//     PlcTask Inputs/GVL_iXlinker.EtherCAT_Master_ATxxxx.Beckhoff_AT1xxx.Beckhoff_AT2xxxEK1122.A_0069_AT2050_0501_0019_AT2050_0501.WcState.InputToggle <-> WcState/InputToggle
//     PlcTask Inputs/GVL_iXlinker.EtherCAT_Master_ATxxxx.Beckhoff_AT1xxx.Beckhoff_AT2xxxEK1122.A_0069_AT2050_0501_0019_AT2050_0501.InfoData.AdsAddr <-> InfoData/AdsAddr
//     PlcTask Inputs/GVL_iXlinker.EtherCAT_Master_ATxxxx.Beckhoff_AT1xxx.Beckhoff_AT2xxxEK1122.A_0069_AT2050_0501_0019_AT2050_0501.InfoData.DcOutputShift <-> InfoData/DcOutputShift
//     PlcTask Inputs/GVL_iXlinker.EtherCAT_Master_ATxxxx.Beckhoff_AT1xxx.Beckhoff_AT2xxxEK1122.A_0069_AT2050_0501_0019_AT2050_0501.InfoData.DcInputShift <-> InfoData/DcInputShift
//     PlcTask Inputs/GVL_iXlinker.EtherCAT_Master_ATxxxx.Beckhoff_AT1xxx.Beckhoff_AT2xxxEK1122.A_0069_AT2050_0501_0019_AT2050_0501.InfoData.State <-> InfoData/State
//   PLC/PLC Instance <-> EtherCAT Master ATxxxx/Beckhoff AT1xxx/Beckhoff AT2xxxEK1122/A_0069(AT2050-0501-0019) (AT2050-0501)/A_0081(AT2002-5250-0018) (AT2002-5250)
//     PlcTask Inputs/GVL_iXlinker.EtherCAT_Master_ATxxxx.Beckhoff_AT1xxx.Beckhoff_AT2xxxEK1122.A_0069_AT2050_0501_0019_AT2050_0501.A_0081_AT2002_5250_0018_AT2002_5250.FB_Inputs.Status <-> FB Inputs/Status
//     PlcTask Inputs/GVL_iXlinker.EtherCAT_Master_ATxxxx.Beckhoff_AT1xxx.Beckhoff_AT2xxxEK1122.A_0069_AT2050_0501_0019_AT2050_0501.A_0081_AT2002_5250_0018_AT2002_5250.FB_Inputs.Value_Channel[0] <-> FB Inputs/Value Channel 01
//     PlcTask Inputs/GVL_iXlinker.EtherCAT_Master_ATxxxx.Beckhoff_AT1xxx.Beckhoff_AT2xxxEK1122.A_0069_AT2050_0501_0019_AT2050_0501.A_0081_AT2002_5250_0018_AT2002_5250.FB_Inputs.Value_Channel[1] <-> FB Inputs/Value Channel 02
//     PlcTask Inputs/GVL_iXlinker.EtherCAT_Master_ATxxxx.Beckhoff_AT1xxx.Beckhoff_AT2xxxEK1122.A_0069_AT2050_0501_0019_AT2050_0501.A_0081_AT2002_5250_0018_AT2002_5250.FB_Inputs.Value_Channel[2] <-> FB Inputs/Value Channel 03
//     PlcTask Inputs/GVL_iXlinker.EtherCAT_Master_ATxxxx.Beckhoff_AT1xxx.Beckhoff_AT2xxxEK1122.A_0069_AT2050_0501_0019_AT2050_0501.A_0081_AT2002_5250_0018_AT2002_5250.FB_Inputs.Value_Channel[3] <-> FB Inputs/Value Channel 04
//     PlcTask Inputs/GVL_iXlinker.EtherCAT_Master_ATxxxx.Beckhoff_AT1xxx.Beckhoff_AT2xxxEK1122.A_0069_AT2050_0501_0019_AT2050_0501.A_0081_AT2002_5250_0018_AT2002_5250.FB_Inputs.Value_Channel[4] <-> FB Inputs/Value Channel 05
//     PlcTask Inputs/GVL_iXlinker.EtherCAT_Master_ATxxxx.Beckhoff_AT1xxx.Beckhoff_AT2xxxEK1122.A_0069_AT2050_0501_0019_AT2050_0501.A_0081_AT2002_5250_0018_AT2002_5250.FB_Inputs.Value_Channel[5] <-> FB Inputs/Value Channel 06
//     PlcTask Inputs/GVL_iXlinker.EtherCAT_Master_ATxxxx.Beckhoff_AT1xxx.Beckhoff_AT2xxxEK1122.A_0069_AT2050_0501_0019_AT2050_0501.A_0081_AT2002_5250_0018_AT2002_5250.FB_Inputs.Value_Channel[6] <-> FB Inputs/Value Channel 07
//     PlcTask Inputs/GVL_iXlinker.EtherCAT_Master_ATxxxx.Beckhoff_AT1xxx.Beckhoff_AT2xxxEK1122.A_0069_AT2050_0501_0019_AT2050_0501.A_0081_AT2002_5250_0018_AT2002_5250.FB_Inputs.Value_Channel[7] <-> FB Inputs/Value Channel 08
//     PlcTask Inputs/GVL_iXlinker.EtherCAT_Master_ATxxxx.Beckhoff_AT1xxx.Beckhoff_AT2xxxEK1122.A_0069_AT2050_0501_0019_AT2050_0501.A_0081_AT2002_5250_0018_AT2002_5250.FB_Inputs.Value_Channel[8] <-> FB Inputs/Value Channel 09
//     PlcTask Inputs/GVL_iXlinker.EtherCAT_Master_ATxxxx.Beckhoff_AT1xxx.Beckhoff_AT2xxxEK1122.A_0069_AT2050_0501_0019_AT2050_0501.A_0081_AT2002_5250_0018_AT2002_5250.FB_Inputs.Value_Channel[9] <-> FB Inputs/Value Channel 10
//     PlcTask Inputs/GVL_iXlinker.EtherCAT_Master_ATxxxx.Beckhoff_AT1xxx.Beckhoff_AT2xxxEK1122.A_0069_AT2050_0501_0019_AT2050_0501.A_0081_AT2002_5250_0018_AT2002_5250.FB_Inputs.Value_Channel[10] <-> FB Inputs/Value Channel 11
//     PlcTask Inputs/GVL_iXlinker.EtherCAT_Master_ATxxxx.Beckhoff_AT1xxx.Beckhoff_AT2xxxEK1122.A_0069_AT2050_0501_0019_AT2050_0501.A_0081_AT2002_5250_0018_AT2002_5250.FB_Inputs.Value_Channel[11] <-> FB Inputs/Value Channel 12
//     PlcTask Inputs/GVL_iXlinker.EtherCAT_Master_ATxxxx.Beckhoff_AT1xxx.Beckhoff_AT2xxxEK1122.A_0069_AT2050_0501_0019_AT2050_0501.A_0081_AT2002_5250_0018_AT2002_5250.FB_Inputs.Value_Channel[12] <-> FB Inputs/Value Channel 13
//     PlcTask Inputs/GVL_iXlinker.EtherCAT_Master_ATxxxx.Beckhoff_AT1xxx.Beckhoff_AT2xxxEK1122.A_0069_AT2050_0501_0019_AT2050_0501.A_0081_AT2002_5250_0018_AT2002_5250.FB_Inputs.Value_Channel[13] <-> FB Inputs/Value Channel 14
//     PlcTask Inputs/GVL_iXlinker.EtherCAT_Master_ATxxxx.Beckhoff_AT1xxx.Beckhoff_AT2xxxEK1122.A_0069_AT2050_0501_0019_AT2050_0501.A_0081_AT2002_5250_0018_AT2002_5250.FB_Inputs.Value_Channel[14] <-> FB Inputs/Value Channel 15
//     PlcTask Inputs/GVL_iXlinker.EtherCAT_Master_ATxxxx.Beckhoff_AT1xxx.Beckhoff_AT2xxxEK1122.A_0069_AT2050_0501_0019_AT2050_0501.A_0081_AT2002_5250_0018_AT2002_5250.FB_Inputs.Value_Channel[15] <-> FB Inputs/Value Channel 16
//     PlcTask Inputs/GVL_iXlinker.EtherCAT_Master_ATxxxx.Beckhoff_AT1xxx.Beckhoff_AT2xxxEK1122.A_0069_AT2050_0501_0019_AT2050_0501.A_0081_AT2002_5250_0018_AT2002_5250.FB_Inputs.Value_Channel[16] <-> FB Inputs/Value Channel 17
//     PlcTask Inputs/GVL_iXlinker.EtherCAT_Master_ATxxxx.Beckhoff_AT1xxx.Beckhoff_AT2xxxEK1122.A_0069_AT2050_0501_0019_AT2050_0501.A_0081_AT2002_5250_0018_AT2002_5250.FB_Inputs.Value_Channel[17] <-> FB Inputs/Value Channel 18
//     PlcTask Inputs/GVL_iXlinker.EtherCAT_Master_ATxxxx.Beckhoff_AT1xxx.Beckhoff_AT2xxxEK1122.A_0069_AT2050_0501_0019_AT2050_0501.A_0081_AT2002_5250_0018_AT2002_5250.FB_Inputs.Value_Channel[18] <-> FB Inputs/Value Channel 19
//     PlcTask Inputs/GVL_iXlinker.EtherCAT_Master_ATxxxx.Beckhoff_AT1xxx.Beckhoff_AT2xxxEK1122.A_0069_AT2050_0501_0019_AT2050_0501.A_0081_AT2002_5250_0018_AT2002_5250.FB_Inputs.Value_Channel[19] <-> FB Inputs/Value Channel 20
//     PlcTask Inputs/GVL_iXlinker.EtherCAT_Master_ATxxxx.Beckhoff_AT1xxx.Beckhoff_AT2xxxEK1122.A_0069_AT2050_0501_0019_AT2050_0501.A_0081_AT2002_5250_0018_AT2002_5250.FB_Inputs.Value_Channel[20] <-> FB Inputs/Value Channel 21
//     PlcTask Inputs/GVL_iXlinker.EtherCAT_Master_ATxxxx.Beckhoff_AT1xxx.Beckhoff_AT2xxxEK1122.A_0069_AT2050_0501_0019_AT2050_0501.A_0081_AT2002_5250_0018_AT2002_5250.FB_Inputs.Value_Channel[21] <-> FB Inputs/Value Channel 22
//     PlcTask Inputs/GVL_iXlinker.EtherCAT_Master_ATxxxx.Beckhoff_AT1xxx.Beckhoff_AT2xxxEK1122.A_0069_AT2050_0501_0019_AT2050_0501.A_0081_AT2002_5250_0018_AT2002_5250.FB_Inputs.Value_Channel[22] <-> FB Inputs/Value Channel 23
//     PlcTask Inputs/GVL_iXlinker.EtherCAT_Master_ATxxxx.Beckhoff_AT1xxx.Beckhoff_AT2xxxEK1122.A_0069_AT2050_0501_0019_AT2050_0501.A_0081_AT2002_5250_0018_AT2002_5250.FB_Inputs.Value_Channel[23] <-> FB Inputs/Value Channel 24
//     PlcTask Inputs/GVL_iXlinker.EtherCAT_Master_ATxxxx.Beckhoff_AT1xxx.Beckhoff_AT2xxxEK1122.A_0069_AT2050_0501_0019_AT2050_0501.A_0081_AT2002_5250_0018_AT2002_5250.FB_Inputs.Value_Channel[24] <-> FB Inputs/Value Channel 25
//     PlcTask Inputs/GVL_iXlinker.EtherCAT_Master_ATxxxx.Beckhoff_AT1xxx.Beckhoff_AT2xxxEK1122.A_0069_AT2050_0501_0019_AT2050_0501.A_0081_AT2002_5250_0018_AT2002_5250.FB_Inputs.Value_Channel[25] <-> FB Inputs/Value Channel 26
//     PlcTask Inputs/GVL_iXlinker.EtherCAT_Master_ATxxxx.Beckhoff_AT1xxx.Beckhoff_AT2xxxEK1122.A_0069_AT2050_0501_0019_AT2050_0501.A_0081_AT2002_5250_0018_AT2002_5250.FB_Inputs.Value_Channel[26] <-> FB Inputs/Value Channel 27
//     PlcTask Inputs/GVL_iXlinker.EtherCAT_Master_ATxxxx.Beckhoff_AT1xxx.Beckhoff_AT2xxxEK1122.A_0069_AT2050_0501_0019_AT2050_0501.A_0081_AT2002_5250_0018_AT2002_5250.FB_Inputs.Value_Channel[27] <-> FB Inputs/Value Channel 28
//     PlcTask Inputs/GVL_iXlinker.EtherCAT_Master_ATxxxx.Beckhoff_AT1xxx.Beckhoff_AT2xxxEK1122.A_0069_AT2050_0501_0019_AT2050_0501.A_0081_AT2002_5250_0018_AT2002_5250.FB_Inputs.Value_Channel[28] <-> FB Inputs/Value Channel 29
//     PlcTask Inputs/GVL_iXlinker.EtherCAT_Master_ATxxxx.Beckhoff_AT1xxx.Beckhoff_AT2xxxEK1122.A_0069_AT2050_0501_0019_AT2050_0501.A_0081_AT2002_5250_0018_AT2002_5250.FB_Inputs.Value_Channel[29] <-> FB Inputs/Value Channel 30
//     PlcTask Inputs/GVL_iXlinker.EtherCAT_Master_ATxxxx.Beckhoff_AT1xxx.Beckhoff_AT2xxxEK1122.A_0069_AT2050_0501_0019_AT2050_0501.A_0081_AT2002_5250_0018_AT2002_5250.FB_Inputs.Value_Channel[30] <-> FB Inputs/Value Channel 31
//     PlcTask Inputs/GVL_iXlinker.EtherCAT_Master_ATxxxx.Beckhoff_AT1xxx.Beckhoff_AT2xxxEK1122.A_0069_AT2050_0501_0019_AT2050_0501.A_0081_AT2002_5250_0018_AT2002_5250.FB_Inputs.Value_Channel[31] <-> FB Inputs/Value Channel 32
//     PlcTask Outputs/GVL_iXlinker.EtherCAT_Master_ATxxxx.Beckhoff_AT1xxx.Beckhoff_AT2xxxEK1122.A_0069_AT2050_0501_0019_AT2050_0501.A_0081_AT2002_5250_0018_AT2002_5250.FB_Outputs.Control <-> FB Outputs/Control
//     PlcTask Inputs/GVL_iXlinker.EtherCAT_Master_ATxxxx.Beckhoff_AT1xxx.Beckhoff_AT2xxxEK1122.A_0069_AT2050_0501_0019_AT2050_0501.A_0081_AT2002_5250_0018_AT2002_5250.WcState.WcState <-> WcState/WcState
//     PlcTask Inputs/GVL_iXlinker.EtherCAT_Master_ATxxxx.Beckhoff_AT1xxx.Beckhoff_AT2xxxEK1122.A_0069_AT2050_0501_0019_AT2050_0501.A_0081_AT2002_5250_0018_AT2002_5250.WcState.InputToggle <-> WcState/InputToggle
//     PlcTask Inputs/GVL_iXlinker.EtherCAT_Master_ATxxxx.Beckhoff_AT1xxx.Beckhoff_AT2xxxEK1122.A_0069_AT2050_0501_0019_AT2050_0501.A_0081_AT2002_5250_0018_AT2002_5250.InfoData.DcOutputShift <-> InfoData/DcOutputShift
//     PlcTask Inputs/GVL_iXlinker.EtherCAT_Master_ATxxxx.Beckhoff_AT1xxx.Beckhoff_AT2xxxEK1122.A_0069_AT2050_0501_0019_AT2050_0501.A_0081_AT2002_5250_0018_AT2002_5250.InfoData.DcInputShift <-> InfoData/DcInputShift
//     PlcTask Inputs/GVL_iXlinker.EtherCAT_Master_ATxxxx.Beckhoff_AT1xxx.Beckhoff_AT2xxxEK1122.A_0069_AT2050_0501_0019_AT2050_0501.A_0081_AT2002_5250_0018_AT2002_5250.InfoData.State <-> InfoData/State
//   PLC/PLC Instance <-> EtherCAT Master ATxxxx/Beckhoff AT1xxx/Beckhoff AT2xxxEK1122/A_0070(AT2050-0501-0022) (AT2050-0501)
//     PlcTask Inputs/GVL_iXlinker.EtherCAT_Master_ATxxxx.Beckhoff_AT1xxx.Beckhoff_AT2xxxEK1122.A_0070_AT2050_0501_0022_AT2050_0501.CC_Inputs.Status <-> CC Inputs/Status
//     PlcTask Inputs/GVL_iXlinker.EtherCAT_Master_ATxxxx.Beckhoff_AT1xxx.Beckhoff_AT2xxxEK1122.A_0070_AT2050_0501_0022_AT2050_0501.CC_Inputs.Current_actual_value_Ch[0] <-> CC Inputs/Current actual value Ch.1
//     PlcTask Inputs/GVL_iXlinker.EtherCAT_Master_ATxxxx.Beckhoff_AT1xxx.Beckhoff_AT2xxxEK1122.A_0070_AT2050_0501_0022_AT2050_0501.CC_Inputs.Current_actual_value_Ch[1] <-> CC Inputs/Current actual value Ch.2
//     PlcTask Inputs/GVL_iXlinker.EtherCAT_Master_ATxxxx.Beckhoff_AT1xxx.Beckhoff_AT2xxxEK1122.A_0070_AT2050_0501_0022_AT2050_0501.CC_Inputs.Current_actual_value_Ch[2] <-> CC Inputs/Current actual value Ch.3
//     PlcTask Inputs/GVL_iXlinker.EtherCAT_Master_ATxxxx.Beckhoff_AT1xxx.Beckhoff_AT2xxxEK1122.A_0070_AT2050_0501_0022_AT2050_0501.CC_Inputs.Current_actual_value_Ch[3] <-> CC Inputs/Current actual value Ch.4
//     PlcTask Inputs/GVL_iXlinker.EtherCAT_Master_ATxxxx.Beckhoff_AT1xxx.Beckhoff_AT2xxxEK1122.A_0070_AT2050_0501_0022_AT2050_0501.CC_Inputs.Current_actual_value_Ch[4] <-> CC Inputs/Current actual value Ch.5
//     PlcTask Inputs/GVL_iXlinker.EtherCAT_Master_ATxxxx.Beckhoff_AT1xxx.Beckhoff_AT2xxxEK1122.A_0070_AT2050_0501_0022_AT2050_0501.CC_Inputs.Current_actual_value_Ch[5] <-> CC Inputs/Current actual value Ch.6
//     PlcTask Inputs/GVL_iXlinker.EtherCAT_Master_ATxxxx.Beckhoff_AT1xxx.Beckhoff_AT2xxxEK1122.A_0070_AT2050_0501_0022_AT2050_0501.CC_Inputs.Current_actual_value_Ch[6] <-> CC Inputs/Current actual value Ch.7
//     PlcTask Inputs/GVL_iXlinker.EtherCAT_Master_ATxxxx.Beckhoff_AT1xxx.Beckhoff_AT2xxxEK1122.A_0070_AT2050_0501_0022_AT2050_0501.CC_Inputs.Current_actual_value_Ch[7] <-> CC Inputs/Current actual value Ch.8
//     PlcTask Inputs/GVL_iXlinker.EtherCAT_Master_ATxxxx.Beckhoff_AT1xxx.Beckhoff_AT2xxxEK1122.A_0070_AT2050_0501_0022_AT2050_0501.CC_Inputs.Current_actual_value_Ch[8] <-> CC Inputs/Current actual value Ch.9
//     PlcTask Inputs/GVL_iXlinker.EtherCAT_Master_ATxxxx.Beckhoff_AT1xxx.Beckhoff_AT2xxxEK1122.A_0070_AT2050_0501_0022_AT2050_0501.CC_Inputs.Current_actual_value_Ch[9] <-> CC Inputs/Current actual value Ch.10
//     PlcTask Inputs/GVL_iXlinker.EtherCAT_Master_ATxxxx.Beckhoff_AT1xxx.Beckhoff_AT2xxxEK1122.A_0070_AT2050_0501_0022_AT2050_0501.CC_Inputs.Current_actual_value_Ch[10] <-> CC Inputs/Current actual value Ch.11
//     PlcTask Inputs/GVL_iXlinker.EtherCAT_Master_ATxxxx.Beckhoff_AT1xxx.Beckhoff_AT2xxxEK1122.A_0070_AT2050_0501_0022_AT2050_0501.CC_Inputs.Current_actual_value_Ch[11] <-> CC Inputs/Current actual value Ch.12
//     PlcTask Inputs/GVL_iXlinker.EtherCAT_Master_ATxxxx.Beckhoff_AT1xxx.Beckhoff_AT2xxxEK1122.A_0070_AT2050_0501_0022_AT2050_0501.CC_Inputs.Current_actual_value_Ch[12] <-> CC Inputs/Current actual value Ch.13
//     PlcTask Inputs/GVL_iXlinker.EtherCAT_Master_ATxxxx.Beckhoff_AT1xxx.Beckhoff_AT2xxxEK1122.A_0070_AT2050_0501_0022_AT2050_0501.CC_Inputs.Current_actual_value_Ch[13] <-> CC Inputs/Current actual value Ch.14
//     PlcTask Inputs/GVL_iXlinker.EtherCAT_Master_ATxxxx.Beckhoff_AT1xxx.Beckhoff_AT2xxxEK1122.A_0070_AT2050_0501_0022_AT2050_0501.CC_Inputs.Current_actual_value_Ch[14] <-> CC Inputs/Current actual value Ch.15
//     PlcTask Outputs/GVL_iXlinker.EtherCAT_Master_ATxxxx.Beckhoff_AT1xxx.Beckhoff_AT2xxxEK1122.A_0070_AT2050_0501_0022_AT2050_0501.CC_Outputs.Control <-> CC Outputs/Control
//     PlcTask Outputs/GVL_iXlinker.EtherCAT_Master_ATxxxx.Beckhoff_AT1xxx.Beckhoff_AT2xxxEK1122.A_0070_AT2050_0501_0022_AT2050_0501.CC_Outputs.Current_setpoint_value_Ch[0] <-> CC Outputs/Current setpoint value Ch.1
//     PlcTask Outputs/GVL_iXlinker.EtherCAT_Master_ATxxxx.Beckhoff_AT1xxx.Beckhoff_AT2xxxEK1122.A_0070_AT2050_0501_0022_AT2050_0501.CC_Outputs.Current_setpoint_value_Ch[1] <-> CC Outputs/Current setpoint value Ch.2
//     PlcTask Outputs/GVL_iXlinker.EtherCAT_Master_ATxxxx.Beckhoff_AT1xxx.Beckhoff_AT2xxxEK1122.A_0070_AT2050_0501_0022_AT2050_0501.CC_Outputs.Current_setpoint_value_Ch[2] <-> CC Outputs/Current setpoint value Ch.3
//     PlcTask Outputs/GVL_iXlinker.EtherCAT_Master_ATxxxx.Beckhoff_AT1xxx.Beckhoff_AT2xxxEK1122.A_0070_AT2050_0501_0022_AT2050_0501.CC_Outputs.Current_setpoint_value_Ch[3] <-> CC Outputs/Current setpoint value Ch.4
//     PlcTask Outputs/GVL_iXlinker.EtherCAT_Master_ATxxxx.Beckhoff_AT1xxx.Beckhoff_AT2xxxEK1122.A_0070_AT2050_0501_0022_AT2050_0501.CC_Outputs.Current_setpoint_value_Ch[4] <-> CC Outputs/Current setpoint value Ch.5
//     PlcTask Outputs/GVL_iXlinker.EtherCAT_Master_ATxxxx.Beckhoff_AT1xxx.Beckhoff_AT2xxxEK1122.A_0070_AT2050_0501_0022_AT2050_0501.CC_Outputs.Current_setpoint_value_Ch[5] <-> CC Outputs/Current setpoint value Ch.6
//     PlcTask Outputs/GVL_iXlinker.EtherCAT_Master_ATxxxx.Beckhoff_AT1xxx.Beckhoff_AT2xxxEK1122.A_0070_AT2050_0501_0022_AT2050_0501.CC_Outputs.Current_setpoint_value_Ch[6] <-> CC Outputs/Current setpoint value Ch.7
//     PlcTask Outputs/GVL_iXlinker.EtherCAT_Master_ATxxxx.Beckhoff_AT1xxx.Beckhoff_AT2xxxEK1122.A_0070_AT2050_0501_0022_AT2050_0501.CC_Outputs.Current_setpoint_value_Ch[7] <-> CC Outputs/Current setpoint value Ch.8
//     PlcTask Outputs/GVL_iXlinker.EtherCAT_Master_ATxxxx.Beckhoff_AT1xxx.Beckhoff_AT2xxxEK1122.A_0070_AT2050_0501_0022_AT2050_0501.CC_Outputs.Current_setpoint_value_Ch[8] <-> CC Outputs/Current setpoint value Ch.9
//     PlcTask Outputs/GVL_iXlinker.EtherCAT_Master_ATxxxx.Beckhoff_AT1xxx.Beckhoff_AT2xxxEK1122.A_0070_AT2050_0501_0022_AT2050_0501.CC_Outputs.Current_setpoint_value_Ch[9] <-> CC Outputs/Current setpoint value Ch.10
//     PlcTask Outputs/GVL_iXlinker.EtherCAT_Master_ATxxxx.Beckhoff_AT1xxx.Beckhoff_AT2xxxEK1122.A_0070_AT2050_0501_0022_AT2050_0501.CC_Outputs.Current_setpoint_value_Ch[10] <-> CC Outputs/Current setpoint value Ch.11
//     PlcTask Outputs/GVL_iXlinker.EtherCAT_Master_ATxxxx.Beckhoff_AT1xxx.Beckhoff_AT2xxxEK1122.A_0070_AT2050_0501_0022_AT2050_0501.CC_Outputs.Current_setpoint_value_Ch[11] <-> CC Outputs/Current setpoint value Ch.12
//     PlcTask Outputs/GVL_iXlinker.EtherCAT_Master_ATxxxx.Beckhoff_AT1xxx.Beckhoff_AT2xxxEK1122.A_0070_AT2050_0501_0022_AT2050_0501.CC_Outputs.Current_setpoint_value_Ch[12] <-> CC Outputs/Current setpoint value Ch.13
//     PlcTask Outputs/GVL_iXlinker.EtherCAT_Master_ATxxxx.Beckhoff_AT1xxx.Beckhoff_AT2xxxEK1122.A_0070_AT2050_0501_0022_AT2050_0501.CC_Outputs.Current_setpoint_value_Ch[13] <-> CC Outputs/Current setpoint value Ch.14
//     PlcTask Outputs/GVL_iXlinker.EtherCAT_Master_ATxxxx.Beckhoff_AT1xxx.Beckhoff_AT2xxxEK1122.A_0070_AT2050_0501_0022_AT2050_0501.CC_Outputs.Current_setpoint_value_Ch[14] <-> CC Outputs/Current setpoint value Ch.15
//     PlcTask Inputs/GVL_iXlinker.EtherCAT_Master_ATxxxx.Beckhoff_AT1xxx.Beckhoff_AT2xxxEK1122.A_0070_AT2050_0501_0022_AT2050_0501.WcState.WcState <-> WcState/WcState
//     PlcTask Inputs/GVL_iXlinker.EtherCAT_Master_ATxxxx.Beckhoff_AT1xxx.Beckhoff_AT2xxxEK1122.A_0070_AT2050_0501_0022_AT2050_0501.WcState.InputToggle <-> WcState/InputToggle
//     PlcTask Inputs/GVL_iXlinker.EtherCAT_Master_ATxxxx.Beckhoff_AT1xxx.Beckhoff_AT2xxxEK1122.A_0070_AT2050_0501_0022_AT2050_0501.InfoData.AdsAddr <-> InfoData/AdsAddr
//     PlcTask Inputs/GVL_iXlinker.EtherCAT_Master_ATxxxx.Beckhoff_AT1xxx.Beckhoff_AT2xxxEK1122.A_0070_AT2050_0501_0022_AT2050_0501.InfoData.DcOutputShift <-> InfoData/DcOutputShift
//     PlcTask Inputs/GVL_iXlinker.EtherCAT_Master_ATxxxx.Beckhoff_AT1xxx.Beckhoff_AT2xxxEK1122.A_0070_AT2050_0501_0022_AT2050_0501.InfoData.DcInputShift <-> InfoData/DcInputShift
//     PlcTask Inputs/GVL_iXlinker.EtherCAT_Master_ATxxxx.Beckhoff_AT1xxx.Beckhoff_AT2xxxEK1122.A_0070_AT2050_0501_0022_AT2050_0501.InfoData.State <-> InfoData/State
//   PLC/PLC Instance <-> EtherCAT Master ATxxxx/Beckhoff AT1xxx/Beckhoff AT2xxxEK1122/A_0070(AT2050-0501-0022) (AT2050-0501)/A_0082(AT2002-5250-0019) (AT2002-5250)
//     PlcTask Inputs/GVL_iXlinker.EtherCAT_Master_ATxxxx.Beckhoff_AT1xxx.Beckhoff_AT2xxxEK1122.A_0070_AT2050_0501_0022_AT2050_0501.A_0082_AT2002_5250_0019_AT2002_5250.FB_Inputs.Status <-> FB Inputs/Status
//     PlcTask Inputs/GVL_iXlinker.EtherCAT_Master_ATxxxx.Beckhoff_AT1xxx.Beckhoff_AT2xxxEK1122.A_0070_AT2050_0501_0022_AT2050_0501.A_0082_AT2002_5250_0019_AT2002_5250.FB_Inputs.Value_Channel[0] <-> FB Inputs/Value Channel 01
//     PlcTask Inputs/GVL_iXlinker.EtherCAT_Master_ATxxxx.Beckhoff_AT1xxx.Beckhoff_AT2xxxEK1122.A_0070_AT2050_0501_0022_AT2050_0501.A_0082_AT2002_5250_0019_AT2002_5250.FB_Inputs.Value_Channel[1] <-> FB Inputs/Value Channel 02
//     PlcTask Inputs/GVL_iXlinker.EtherCAT_Master_ATxxxx.Beckhoff_AT1xxx.Beckhoff_AT2xxxEK1122.A_0070_AT2050_0501_0022_AT2050_0501.A_0082_AT2002_5250_0019_AT2002_5250.FB_Inputs.Value_Channel[2] <-> FB Inputs/Value Channel 03
//     PlcTask Inputs/GVL_iXlinker.EtherCAT_Master_ATxxxx.Beckhoff_AT1xxx.Beckhoff_AT2xxxEK1122.A_0070_AT2050_0501_0022_AT2050_0501.A_0082_AT2002_5250_0019_AT2002_5250.FB_Inputs.Value_Channel[3] <-> FB Inputs/Value Channel 04
//     PlcTask Inputs/GVL_iXlinker.EtherCAT_Master_ATxxxx.Beckhoff_AT1xxx.Beckhoff_AT2xxxEK1122.A_0070_AT2050_0501_0022_AT2050_0501.A_0082_AT2002_5250_0019_AT2002_5250.FB_Inputs.Value_Channel[4] <-> FB Inputs/Value Channel 05
//     PlcTask Inputs/GVL_iXlinker.EtherCAT_Master_ATxxxx.Beckhoff_AT1xxx.Beckhoff_AT2xxxEK1122.A_0070_AT2050_0501_0022_AT2050_0501.A_0082_AT2002_5250_0019_AT2002_5250.FB_Inputs.Value_Channel[5] <-> FB Inputs/Value Channel 06
//     PlcTask Inputs/GVL_iXlinker.EtherCAT_Master_ATxxxx.Beckhoff_AT1xxx.Beckhoff_AT2xxxEK1122.A_0070_AT2050_0501_0022_AT2050_0501.A_0082_AT2002_5250_0019_AT2002_5250.FB_Inputs.Value_Channel[6] <-> FB Inputs/Value Channel 07
//     PlcTask Inputs/GVL_iXlinker.EtherCAT_Master_ATxxxx.Beckhoff_AT1xxx.Beckhoff_AT2xxxEK1122.A_0070_AT2050_0501_0022_AT2050_0501.A_0082_AT2002_5250_0019_AT2002_5250.FB_Inputs.Value_Channel[7] <-> FB Inputs/Value Channel 08
//     PlcTask Inputs/GVL_iXlinker.EtherCAT_Master_ATxxxx.Beckhoff_AT1xxx.Beckhoff_AT2xxxEK1122.A_0070_AT2050_0501_0022_AT2050_0501.A_0082_AT2002_5250_0019_AT2002_5250.FB_Inputs.Value_Channel[8] <-> FB Inputs/Value Channel 09
//     PlcTask Inputs/GVL_iXlinker.EtherCAT_Master_ATxxxx.Beckhoff_AT1xxx.Beckhoff_AT2xxxEK1122.A_0070_AT2050_0501_0022_AT2050_0501.A_0082_AT2002_5250_0019_AT2002_5250.FB_Inputs.Value_Channel[9] <-> FB Inputs/Value Channel 10
//     PlcTask Inputs/GVL_iXlinker.EtherCAT_Master_ATxxxx.Beckhoff_AT1xxx.Beckhoff_AT2xxxEK1122.A_0070_AT2050_0501_0022_AT2050_0501.A_0082_AT2002_5250_0019_AT2002_5250.FB_Inputs.Value_Channel[10] <-> FB Inputs/Value Channel 11
//     PlcTask Inputs/GVL_iXlinker.EtherCAT_Master_ATxxxx.Beckhoff_AT1xxx.Beckhoff_AT2xxxEK1122.A_0070_AT2050_0501_0022_AT2050_0501.A_0082_AT2002_5250_0019_AT2002_5250.FB_Inputs.Value_Channel[11] <-> FB Inputs/Value Channel 12
//     PlcTask Inputs/GVL_iXlinker.EtherCAT_Master_ATxxxx.Beckhoff_AT1xxx.Beckhoff_AT2xxxEK1122.A_0070_AT2050_0501_0022_AT2050_0501.A_0082_AT2002_5250_0019_AT2002_5250.FB_Inputs.Value_Channel[12] <-> FB Inputs/Value Channel 13
//     PlcTask Inputs/GVL_iXlinker.EtherCAT_Master_ATxxxx.Beckhoff_AT1xxx.Beckhoff_AT2xxxEK1122.A_0070_AT2050_0501_0022_AT2050_0501.A_0082_AT2002_5250_0019_AT2002_5250.FB_Inputs.Value_Channel[13] <-> FB Inputs/Value Channel 14
//     PlcTask Inputs/GVL_iXlinker.EtherCAT_Master_ATxxxx.Beckhoff_AT1xxx.Beckhoff_AT2xxxEK1122.A_0070_AT2050_0501_0022_AT2050_0501.A_0082_AT2002_5250_0019_AT2002_5250.FB_Inputs.Value_Channel[14] <-> FB Inputs/Value Channel 15
//     PlcTask Inputs/GVL_iXlinker.EtherCAT_Master_ATxxxx.Beckhoff_AT1xxx.Beckhoff_AT2xxxEK1122.A_0070_AT2050_0501_0022_AT2050_0501.A_0082_AT2002_5250_0019_AT2002_5250.FB_Inputs.Value_Channel[15] <-> FB Inputs/Value Channel 16
//     PlcTask Inputs/GVL_iXlinker.EtherCAT_Master_ATxxxx.Beckhoff_AT1xxx.Beckhoff_AT2xxxEK1122.A_0070_AT2050_0501_0022_AT2050_0501.A_0082_AT2002_5250_0019_AT2002_5250.FB_Inputs.Value_Channel[16] <-> FB Inputs/Value Channel 17
//     PlcTask Inputs/GVL_iXlinker.EtherCAT_Master_ATxxxx.Beckhoff_AT1xxx.Beckhoff_AT2xxxEK1122.A_0070_AT2050_0501_0022_AT2050_0501.A_0082_AT2002_5250_0019_AT2002_5250.FB_Inputs.Value_Channel[17] <-> FB Inputs/Value Channel 18
//     PlcTask Inputs/GVL_iXlinker.EtherCAT_Master_ATxxxx.Beckhoff_AT1xxx.Beckhoff_AT2xxxEK1122.A_0070_AT2050_0501_0022_AT2050_0501.A_0082_AT2002_5250_0019_AT2002_5250.FB_Inputs.Value_Channel[18] <-> FB Inputs/Value Channel 19
//     PlcTask Inputs/GVL_iXlinker.EtherCAT_Master_ATxxxx.Beckhoff_AT1xxx.Beckhoff_AT2xxxEK1122.A_0070_AT2050_0501_0022_AT2050_0501.A_0082_AT2002_5250_0019_AT2002_5250.FB_Inputs.Value_Channel[19] <-> FB Inputs/Value Channel 20
//     PlcTask Inputs/GVL_iXlinker.EtherCAT_Master_ATxxxx.Beckhoff_AT1xxx.Beckhoff_AT2xxxEK1122.A_0070_AT2050_0501_0022_AT2050_0501.A_0082_AT2002_5250_0019_AT2002_5250.FB_Inputs.Value_Channel[20] <-> FB Inputs/Value Channel 21
//     PlcTask Inputs/GVL_iXlinker.EtherCAT_Master_ATxxxx.Beckhoff_AT1xxx.Beckhoff_AT2xxxEK1122.A_0070_AT2050_0501_0022_AT2050_0501.A_0082_AT2002_5250_0019_AT2002_5250.FB_Inputs.Value_Channel[21] <-> FB Inputs/Value Channel 22
//     PlcTask Inputs/GVL_iXlinker.EtherCAT_Master_ATxxxx.Beckhoff_AT1xxx.Beckhoff_AT2xxxEK1122.A_0070_AT2050_0501_0022_AT2050_0501.A_0082_AT2002_5250_0019_AT2002_5250.FB_Inputs.Value_Channel[22] <-> FB Inputs/Value Channel 23
//     PlcTask Inputs/GVL_iXlinker.EtherCAT_Master_ATxxxx.Beckhoff_AT1xxx.Beckhoff_AT2xxxEK1122.A_0070_AT2050_0501_0022_AT2050_0501.A_0082_AT2002_5250_0019_AT2002_5250.FB_Inputs.Value_Channel[23] <-> FB Inputs/Value Channel 24
//     PlcTask Inputs/GVL_iXlinker.EtherCAT_Master_ATxxxx.Beckhoff_AT1xxx.Beckhoff_AT2xxxEK1122.A_0070_AT2050_0501_0022_AT2050_0501.A_0082_AT2002_5250_0019_AT2002_5250.FB_Inputs.Value_Channel[24] <-> FB Inputs/Value Channel 25
//     PlcTask Inputs/GVL_iXlinker.EtherCAT_Master_ATxxxx.Beckhoff_AT1xxx.Beckhoff_AT2xxxEK1122.A_0070_AT2050_0501_0022_AT2050_0501.A_0082_AT2002_5250_0019_AT2002_5250.FB_Inputs.Value_Channel[25] <-> FB Inputs/Value Channel 26
//     PlcTask Inputs/GVL_iXlinker.EtherCAT_Master_ATxxxx.Beckhoff_AT1xxx.Beckhoff_AT2xxxEK1122.A_0070_AT2050_0501_0022_AT2050_0501.A_0082_AT2002_5250_0019_AT2002_5250.FB_Inputs.Value_Channel[26] <-> FB Inputs/Value Channel 27
//     PlcTask Inputs/GVL_iXlinker.EtherCAT_Master_ATxxxx.Beckhoff_AT1xxx.Beckhoff_AT2xxxEK1122.A_0070_AT2050_0501_0022_AT2050_0501.A_0082_AT2002_5250_0019_AT2002_5250.FB_Inputs.Value_Channel[27] <-> FB Inputs/Value Channel 28
//     PlcTask Inputs/GVL_iXlinker.EtherCAT_Master_ATxxxx.Beckhoff_AT1xxx.Beckhoff_AT2xxxEK1122.A_0070_AT2050_0501_0022_AT2050_0501.A_0082_AT2002_5250_0019_AT2002_5250.FB_Inputs.Value_Channel[28] <-> FB Inputs/Value Channel 29
//     PlcTask Inputs/GVL_iXlinker.EtherCAT_Master_ATxxxx.Beckhoff_AT1xxx.Beckhoff_AT2xxxEK1122.A_0070_AT2050_0501_0022_AT2050_0501.A_0082_AT2002_5250_0019_AT2002_5250.FB_Inputs.Value_Channel[29] <-> FB Inputs/Value Channel 30
//     PlcTask Inputs/GVL_iXlinker.EtherCAT_Master_ATxxxx.Beckhoff_AT1xxx.Beckhoff_AT2xxxEK1122.A_0070_AT2050_0501_0022_AT2050_0501.A_0082_AT2002_5250_0019_AT2002_5250.FB_Inputs.Value_Channel[30] <-> FB Inputs/Value Channel 31
//     PlcTask Inputs/GVL_iXlinker.EtherCAT_Master_ATxxxx.Beckhoff_AT1xxx.Beckhoff_AT2xxxEK1122.A_0070_AT2050_0501_0022_AT2050_0501.A_0082_AT2002_5250_0019_AT2002_5250.FB_Inputs.Value_Channel[31] <-> FB Inputs/Value Channel 32
//     PlcTask Outputs/GVL_iXlinker.EtherCAT_Master_ATxxxx.Beckhoff_AT1xxx.Beckhoff_AT2xxxEK1122.A_0070_AT2050_0501_0022_AT2050_0501.A_0082_AT2002_5250_0019_AT2002_5250.FB_Outputs.Control <-> FB Outputs/Control
//     PlcTask Inputs/GVL_iXlinker.EtherCAT_Master_ATxxxx.Beckhoff_AT1xxx.Beckhoff_AT2xxxEK1122.A_0070_AT2050_0501_0022_AT2050_0501.A_0082_AT2002_5250_0019_AT2002_5250.WcState.WcState <-> WcState/WcState
//     PlcTask Inputs/GVL_iXlinker.EtherCAT_Master_ATxxxx.Beckhoff_AT1xxx.Beckhoff_AT2xxxEK1122.A_0070_AT2050_0501_0022_AT2050_0501.A_0082_AT2002_5250_0019_AT2002_5250.WcState.InputToggle <-> WcState/InputToggle
//     PlcTask Inputs/GVL_iXlinker.EtherCAT_Master_ATxxxx.Beckhoff_AT1xxx.Beckhoff_AT2xxxEK1122.A_0070_AT2050_0501_0022_AT2050_0501.A_0082_AT2002_5250_0019_AT2002_5250.InfoData.DcOutputShift <-> InfoData/DcOutputShift
//     PlcTask Inputs/GVL_iXlinker.EtherCAT_Master_ATxxxx.Beckhoff_AT1xxx.Beckhoff_AT2xxxEK1122.A_0070_AT2050_0501_0022_AT2050_0501.A_0082_AT2002_5250_0019_AT2002_5250.InfoData.DcInputShift <-> InfoData/DcInputShift
//     PlcTask Inputs/GVL_iXlinker.EtherCAT_Master_ATxxxx.Beckhoff_AT1xxx.Beckhoff_AT2xxxEK1122.A_0070_AT2050_0501_0022_AT2050_0501.A_0082_AT2002_5250_0019_AT2002_5250.InfoData.State <-> InfoData/State
//   PLC/PLC Instance <-> EtherCAT Master ATxxxx/Beckhoff AT1xxx/Beckhoff AT2xxxEK1122/A_0071(AT2050-0501-0023) (AT2050-0501)
//     PlcTask Inputs/GVL_iXlinker.EtherCAT_Master_ATxxxx.Beckhoff_AT1xxx.Beckhoff_AT2xxxEK1122.A_0071_AT2050_0501_0023_AT2050_0501.CC_Inputs.Status <-> CC Inputs/Status
//     PlcTask Inputs/GVL_iXlinker.EtherCAT_Master_ATxxxx.Beckhoff_AT1xxx.Beckhoff_AT2xxxEK1122.A_0071_AT2050_0501_0023_AT2050_0501.CC_Inputs.Current_actual_value_Ch[0] <-> CC Inputs/Current actual value Ch.1
//     PlcTask Inputs/GVL_iXlinker.EtherCAT_Master_ATxxxx.Beckhoff_AT1xxx.Beckhoff_AT2xxxEK1122.A_0071_AT2050_0501_0023_AT2050_0501.CC_Inputs.Current_actual_value_Ch[1] <-> CC Inputs/Current actual value Ch.2
//     PlcTask Inputs/GVL_iXlinker.EtherCAT_Master_ATxxxx.Beckhoff_AT1xxx.Beckhoff_AT2xxxEK1122.A_0071_AT2050_0501_0023_AT2050_0501.CC_Inputs.Current_actual_value_Ch[2] <-> CC Inputs/Current actual value Ch.3
//     PlcTask Inputs/GVL_iXlinker.EtherCAT_Master_ATxxxx.Beckhoff_AT1xxx.Beckhoff_AT2xxxEK1122.A_0071_AT2050_0501_0023_AT2050_0501.CC_Inputs.Current_actual_value_Ch[3] <-> CC Inputs/Current actual value Ch.4
//     PlcTask Inputs/GVL_iXlinker.EtherCAT_Master_ATxxxx.Beckhoff_AT1xxx.Beckhoff_AT2xxxEK1122.A_0071_AT2050_0501_0023_AT2050_0501.CC_Inputs.Current_actual_value_Ch[4] <-> CC Inputs/Current actual value Ch.5
//     PlcTask Inputs/GVL_iXlinker.EtherCAT_Master_ATxxxx.Beckhoff_AT1xxx.Beckhoff_AT2xxxEK1122.A_0071_AT2050_0501_0023_AT2050_0501.CC_Inputs.Current_actual_value_Ch[5] <-> CC Inputs/Current actual value Ch.6
//     PlcTask Inputs/GVL_iXlinker.EtherCAT_Master_ATxxxx.Beckhoff_AT1xxx.Beckhoff_AT2xxxEK1122.A_0071_AT2050_0501_0023_AT2050_0501.CC_Inputs.Current_actual_value_Ch[6] <-> CC Inputs/Current actual value Ch.7
//     PlcTask Inputs/GVL_iXlinker.EtherCAT_Master_ATxxxx.Beckhoff_AT1xxx.Beckhoff_AT2xxxEK1122.A_0071_AT2050_0501_0023_AT2050_0501.CC_Inputs.Current_actual_value_Ch[7] <-> CC Inputs/Current actual value Ch.8
//     PlcTask Inputs/GVL_iXlinker.EtherCAT_Master_ATxxxx.Beckhoff_AT1xxx.Beckhoff_AT2xxxEK1122.A_0071_AT2050_0501_0023_AT2050_0501.CC_Inputs.Current_actual_value_Ch[8] <-> CC Inputs/Current actual value Ch.9
//     PlcTask Inputs/GVL_iXlinker.EtherCAT_Master_ATxxxx.Beckhoff_AT1xxx.Beckhoff_AT2xxxEK1122.A_0071_AT2050_0501_0023_AT2050_0501.CC_Inputs.Current_actual_value_Ch[9] <-> CC Inputs/Current actual value Ch.10
//     PlcTask Inputs/GVL_iXlinker.EtherCAT_Master_ATxxxx.Beckhoff_AT1xxx.Beckhoff_AT2xxxEK1122.A_0071_AT2050_0501_0023_AT2050_0501.CC_Inputs.Current_actual_value_Ch[10] <-> CC Inputs/Current actual value Ch.11
//     PlcTask Inputs/GVL_iXlinker.EtherCAT_Master_ATxxxx.Beckhoff_AT1xxx.Beckhoff_AT2xxxEK1122.A_0071_AT2050_0501_0023_AT2050_0501.CC_Inputs.Current_actual_value_Ch[11] <-> CC Inputs/Current actual value Ch.12
//     PlcTask Inputs/GVL_iXlinker.EtherCAT_Master_ATxxxx.Beckhoff_AT1xxx.Beckhoff_AT2xxxEK1122.A_0071_AT2050_0501_0023_AT2050_0501.CC_Inputs.Current_actual_value_Ch[12] <-> CC Inputs/Current actual value Ch.13
//     PlcTask Inputs/GVL_iXlinker.EtherCAT_Master_ATxxxx.Beckhoff_AT1xxx.Beckhoff_AT2xxxEK1122.A_0071_AT2050_0501_0023_AT2050_0501.CC_Inputs.Current_actual_value_Ch[13] <-> CC Inputs/Current actual value Ch.14
//     PlcTask Inputs/GVL_iXlinker.EtherCAT_Master_ATxxxx.Beckhoff_AT1xxx.Beckhoff_AT2xxxEK1122.A_0071_AT2050_0501_0023_AT2050_0501.CC_Inputs.Current_actual_value_Ch[14] <-> CC Inputs/Current actual value Ch.15
//     PlcTask Outputs/GVL_iXlinker.EtherCAT_Master_ATxxxx.Beckhoff_AT1xxx.Beckhoff_AT2xxxEK1122.A_0071_AT2050_0501_0023_AT2050_0501.CC_Outputs.Control <-> CC Outputs/Control
//     PlcTask Outputs/GVL_iXlinker.EtherCAT_Master_ATxxxx.Beckhoff_AT1xxx.Beckhoff_AT2xxxEK1122.A_0071_AT2050_0501_0023_AT2050_0501.CC_Outputs.Current_setpoint_value_Ch[0] <-> CC Outputs/Current setpoint value Ch.1
//     PlcTask Outputs/GVL_iXlinker.EtherCAT_Master_ATxxxx.Beckhoff_AT1xxx.Beckhoff_AT2xxxEK1122.A_0071_AT2050_0501_0023_AT2050_0501.CC_Outputs.Current_setpoint_value_Ch[1] <-> CC Outputs/Current setpoint value Ch.2
//     PlcTask Outputs/GVL_iXlinker.EtherCAT_Master_ATxxxx.Beckhoff_AT1xxx.Beckhoff_AT2xxxEK1122.A_0071_AT2050_0501_0023_AT2050_0501.CC_Outputs.Current_setpoint_value_Ch[2] <-> CC Outputs/Current setpoint value Ch.3
//     PlcTask Outputs/GVL_iXlinker.EtherCAT_Master_ATxxxx.Beckhoff_AT1xxx.Beckhoff_AT2xxxEK1122.A_0071_AT2050_0501_0023_AT2050_0501.CC_Outputs.Current_setpoint_value_Ch[3] <-> CC Outputs/Current setpoint value Ch.4
//     PlcTask Outputs/GVL_iXlinker.EtherCAT_Master_ATxxxx.Beckhoff_AT1xxx.Beckhoff_AT2xxxEK1122.A_0071_AT2050_0501_0023_AT2050_0501.CC_Outputs.Current_setpoint_value_Ch[4] <-> CC Outputs/Current setpoint value Ch.5
//     PlcTask Outputs/GVL_iXlinker.EtherCAT_Master_ATxxxx.Beckhoff_AT1xxx.Beckhoff_AT2xxxEK1122.A_0071_AT2050_0501_0023_AT2050_0501.CC_Outputs.Current_setpoint_value_Ch[5] <-> CC Outputs/Current setpoint value Ch.6
//     PlcTask Outputs/GVL_iXlinker.EtherCAT_Master_ATxxxx.Beckhoff_AT1xxx.Beckhoff_AT2xxxEK1122.A_0071_AT2050_0501_0023_AT2050_0501.CC_Outputs.Current_setpoint_value_Ch[6] <-> CC Outputs/Current setpoint value Ch.7
//     PlcTask Outputs/GVL_iXlinker.EtherCAT_Master_ATxxxx.Beckhoff_AT1xxx.Beckhoff_AT2xxxEK1122.A_0071_AT2050_0501_0023_AT2050_0501.CC_Outputs.Current_setpoint_value_Ch[7] <-> CC Outputs/Current setpoint value Ch.8
//     PlcTask Outputs/GVL_iXlinker.EtherCAT_Master_ATxxxx.Beckhoff_AT1xxx.Beckhoff_AT2xxxEK1122.A_0071_AT2050_0501_0023_AT2050_0501.CC_Outputs.Current_setpoint_value_Ch[8] <-> CC Outputs/Current setpoint value Ch.9
//     PlcTask Outputs/GVL_iXlinker.EtherCAT_Master_ATxxxx.Beckhoff_AT1xxx.Beckhoff_AT2xxxEK1122.A_0071_AT2050_0501_0023_AT2050_0501.CC_Outputs.Current_setpoint_value_Ch[9] <-> CC Outputs/Current setpoint value Ch.10
//     PlcTask Outputs/GVL_iXlinker.EtherCAT_Master_ATxxxx.Beckhoff_AT1xxx.Beckhoff_AT2xxxEK1122.A_0071_AT2050_0501_0023_AT2050_0501.CC_Outputs.Current_setpoint_value_Ch[10] <-> CC Outputs/Current setpoint value Ch.11
//     PlcTask Outputs/GVL_iXlinker.EtherCAT_Master_ATxxxx.Beckhoff_AT1xxx.Beckhoff_AT2xxxEK1122.A_0071_AT2050_0501_0023_AT2050_0501.CC_Outputs.Current_setpoint_value_Ch[11] <-> CC Outputs/Current setpoint value Ch.12
//     PlcTask Outputs/GVL_iXlinker.EtherCAT_Master_ATxxxx.Beckhoff_AT1xxx.Beckhoff_AT2xxxEK1122.A_0071_AT2050_0501_0023_AT2050_0501.CC_Outputs.Current_setpoint_value_Ch[12] <-> CC Outputs/Current setpoint value Ch.13
//     PlcTask Outputs/GVL_iXlinker.EtherCAT_Master_ATxxxx.Beckhoff_AT1xxx.Beckhoff_AT2xxxEK1122.A_0071_AT2050_0501_0023_AT2050_0501.CC_Outputs.Current_setpoint_value_Ch[13] <-> CC Outputs/Current setpoint value Ch.14
//     PlcTask Outputs/GVL_iXlinker.EtherCAT_Master_ATxxxx.Beckhoff_AT1xxx.Beckhoff_AT2xxxEK1122.A_0071_AT2050_0501_0023_AT2050_0501.CC_Outputs.Current_setpoint_value_Ch[14] <-> CC Outputs/Current setpoint value Ch.15
//     PlcTask Inputs/GVL_iXlinker.EtherCAT_Master_ATxxxx.Beckhoff_AT1xxx.Beckhoff_AT2xxxEK1122.A_0071_AT2050_0501_0023_AT2050_0501.WcState.WcState <-> WcState/WcState
//     PlcTask Inputs/GVL_iXlinker.EtherCAT_Master_ATxxxx.Beckhoff_AT1xxx.Beckhoff_AT2xxxEK1122.A_0071_AT2050_0501_0023_AT2050_0501.WcState.InputToggle <-> WcState/InputToggle
//     PlcTask Inputs/GVL_iXlinker.EtherCAT_Master_ATxxxx.Beckhoff_AT1xxx.Beckhoff_AT2xxxEK1122.A_0071_AT2050_0501_0023_AT2050_0501.InfoData.AdsAddr <-> InfoData/AdsAddr
//     PlcTask Inputs/GVL_iXlinker.EtherCAT_Master_ATxxxx.Beckhoff_AT1xxx.Beckhoff_AT2xxxEK1122.A_0071_AT2050_0501_0023_AT2050_0501.InfoData.DcOutputShift <-> InfoData/DcOutputShift
//     PlcTask Inputs/GVL_iXlinker.EtherCAT_Master_ATxxxx.Beckhoff_AT1xxx.Beckhoff_AT2xxxEK1122.A_0071_AT2050_0501_0023_AT2050_0501.InfoData.DcInputShift <-> InfoData/DcInputShift
//     PlcTask Inputs/GVL_iXlinker.EtherCAT_Master_ATxxxx.Beckhoff_AT1xxx.Beckhoff_AT2xxxEK1122.A_0071_AT2050_0501_0023_AT2050_0501.InfoData.State <-> InfoData/State
//   PLC/PLC Instance <-> EtherCAT Master ATxxxx/Beckhoff AT1xxx/Beckhoff AT2xxxEK1122/A_0071(AT2050-0501-0023) (AT2050-0501)/A_0083(AT2050-5500-0016) (AT2050-5500)
//     PlcTask Inputs/GVL_iXlinker.EtherCAT_Master_ATxxxx.Beckhoff_AT1xxx.Beckhoff_AT2xxxEK1122.A_0071_AT2050_0501_0023_AT2050_0501.A_0083_AT2050_5500_0016_AT2050_5500.FB_Inputs.Status <-> FB Inputs/Status
//     PlcTask Inputs/GVL_iXlinker.EtherCAT_Master_ATxxxx.Beckhoff_AT1xxx.Beckhoff_AT2xxxEK1122.A_0071_AT2050_0501_0023_AT2050_0501.A_0083_AT2050_5500_0016_AT2050_5500.FB_Inputs.Value_Channel[0] <-> FB Inputs/Value Channel 01
//     PlcTask Inputs/GVL_iXlinker.EtherCAT_Master_ATxxxx.Beckhoff_AT1xxx.Beckhoff_AT2xxxEK1122.A_0071_AT2050_0501_0023_AT2050_0501.A_0083_AT2050_5500_0016_AT2050_5500.FB_Inputs.Value_Channel[1] <-> FB Inputs/Value Channel 02
//     PlcTask Inputs/GVL_iXlinker.EtherCAT_Master_ATxxxx.Beckhoff_AT1xxx.Beckhoff_AT2xxxEK1122.A_0071_AT2050_0501_0023_AT2050_0501.A_0083_AT2050_5500_0016_AT2050_5500.FB_Inputs.Value_Channel[2] <-> FB Inputs/Value Channel 03
//     PlcTask Inputs/GVL_iXlinker.EtherCAT_Master_ATxxxx.Beckhoff_AT1xxx.Beckhoff_AT2xxxEK1122.A_0071_AT2050_0501_0023_AT2050_0501.A_0083_AT2050_5500_0016_AT2050_5500.FB_Inputs.Value_Channel[3] <-> FB Inputs/Value Channel 04
//     PlcTask Inputs/GVL_iXlinker.EtherCAT_Master_ATxxxx.Beckhoff_AT1xxx.Beckhoff_AT2xxxEK1122.A_0071_AT2050_0501_0023_AT2050_0501.A_0083_AT2050_5500_0016_AT2050_5500.FB_Inputs.Value_Channel[4] <-> FB Inputs/Value Channel 05
//     PlcTask Inputs/GVL_iXlinker.EtherCAT_Master_ATxxxx.Beckhoff_AT1xxx.Beckhoff_AT2xxxEK1122.A_0071_AT2050_0501_0023_AT2050_0501.A_0083_AT2050_5500_0016_AT2050_5500.FB_Inputs.Value_Channel[5] <-> FB Inputs/Value Channel 06
//     PlcTask Inputs/GVL_iXlinker.EtherCAT_Master_ATxxxx.Beckhoff_AT1xxx.Beckhoff_AT2xxxEK1122.A_0071_AT2050_0501_0023_AT2050_0501.A_0083_AT2050_5500_0016_AT2050_5500.FB_Inputs.Value_Channel[6] <-> FB Inputs/Value Channel 07
//     PlcTask Inputs/GVL_iXlinker.EtherCAT_Master_ATxxxx.Beckhoff_AT1xxx.Beckhoff_AT2xxxEK1122.A_0071_AT2050_0501_0023_AT2050_0501.A_0083_AT2050_5500_0016_AT2050_5500.FB_Inputs.Value_Channel[7] <-> FB Inputs/Value Channel 08
//     PlcTask Inputs/GVL_iXlinker.EtherCAT_Master_ATxxxx.Beckhoff_AT1xxx.Beckhoff_AT2xxxEK1122.A_0071_AT2050_0501_0023_AT2050_0501.A_0083_AT2050_5500_0016_AT2050_5500.FB_Inputs.Value_Channel[8] <-> FB Inputs/Value Channel 09
//     PlcTask Inputs/GVL_iXlinker.EtherCAT_Master_ATxxxx.Beckhoff_AT1xxx.Beckhoff_AT2xxxEK1122.A_0071_AT2050_0501_0023_AT2050_0501.A_0083_AT2050_5500_0016_AT2050_5500.FB_Inputs.Value_Channel[9] <-> FB Inputs/Value Channel 10
//     PlcTask Inputs/GVL_iXlinker.EtherCAT_Master_ATxxxx.Beckhoff_AT1xxx.Beckhoff_AT2xxxEK1122.A_0071_AT2050_0501_0023_AT2050_0501.A_0083_AT2050_5500_0016_AT2050_5500.FB_Inputs.Value_Channel[10] <-> FB Inputs/Value Channel 11
//     PlcTask Inputs/GVL_iXlinker.EtherCAT_Master_ATxxxx.Beckhoff_AT1xxx.Beckhoff_AT2xxxEK1122.A_0071_AT2050_0501_0023_AT2050_0501.A_0083_AT2050_5500_0016_AT2050_5500.FB_Inputs.Value_Channel[11] <-> FB Inputs/Value Channel 12
//     PlcTask Inputs/GVL_iXlinker.EtherCAT_Master_ATxxxx.Beckhoff_AT1xxx.Beckhoff_AT2xxxEK1122.A_0071_AT2050_0501_0023_AT2050_0501.A_0083_AT2050_5500_0016_AT2050_5500.FB_Inputs.Value_Channel[12] <-> FB Inputs/Value Channel 13
//     PlcTask Inputs/GVL_iXlinker.EtherCAT_Master_ATxxxx.Beckhoff_AT1xxx.Beckhoff_AT2xxxEK1122.A_0071_AT2050_0501_0023_AT2050_0501.A_0083_AT2050_5500_0016_AT2050_5500.FB_Inputs.Value_Channel[13] <-> FB Inputs/Value Channel 14
//     PlcTask Inputs/GVL_iXlinker.EtherCAT_Master_ATxxxx.Beckhoff_AT1xxx.Beckhoff_AT2xxxEK1122.A_0071_AT2050_0501_0023_AT2050_0501.A_0083_AT2050_5500_0016_AT2050_5500.FB_Inputs.Value_Channel[14] <-> FB Inputs/Value Channel 15
//     PlcTask Inputs/GVL_iXlinker.EtherCAT_Master_ATxxxx.Beckhoff_AT1xxx.Beckhoff_AT2xxxEK1122.A_0071_AT2050_0501_0023_AT2050_0501.A_0083_AT2050_5500_0016_AT2050_5500.FB_Inputs.Value_Channel[15] <-> FB Inputs/Value Channel 16
//     PlcTask Inputs/GVL_iXlinker.EtherCAT_Master_ATxxxx.Beckhoff_AT1xxx.Beckhoff_AT2xxxEK1122.A_0071_AT2050_0501_0023_AT2050_0501.A_0083_AT2050_5500_0016_AT2050_5500.FB_Inputs.Value_Channel[16] <-> FB Inputs/Value Channel 17
//     PlcTask Inputs/GVL_iXlinker.EtherCAT_Master_ATxxxx.Beckhoff_AT1xxx.Beckhoff_AT2xxxEK1122.A_0071_AT2050_0501_0023_AT2050_0501.A_0083_AT2050_5500_0016_AT2050_5500.FB_Inputs.Value_Channel[17] <-> FB Inputs/Value Channel 18
//     PlcTask Inputs/GVL_iXlinker.EtherCAT_Master_ATxxxx.Beckhoff_AT1xxx.Beckhoff_AT2xxxEK1122.A_0071_AT2050_0501_0023_AT2050_0501.A_0083_AT2050_5500_0016_AT2050_5500.FB_Inputs.Value_Channel[18] <-> FB Inputs/Value Channel 19
//     PlcTask Inputs/GVL_iXlinker.EtherCAT_Master_ATxxxx.Beckhoff_AT1xxx.Beckhoff_AT2xxxEK1122.A_0071_AT2050_0501_0023_AT2050_0501.A_0083_AT2050_5500_0016_AT2050_5500.FB_Inputs.Value_Channel[19] <-> FB Inputs/Value Channel 20
//     PlcTask Inputs/GVL_iXlinker.EtherCAT_Master_ATxxxx.Beckhoff_AT1xxx.Beckhoff_AT2xxxEK1122.A_0071_AT2050_0501_0023_AT2050_0501.A_0083_AT2050_5500_0016_AT2050_5500.FB_Inputs.Value_Channel[20] <-> FB Inputs/Value Channel 21
//     PlcTask Inputs/GVL_iXlinker.EtherCAT_Master_ATxxxx.Beckhoff_AT1xxx.Beckhoff_AT2xxxEK1122.A_0071_AT2050_0501_0023_AT2050_0501.A_0083_AT2050_5500_0016_AT2050_5500.FB_Inputs.Value_Channel[21] <-> FB Inputs/Value Channel 22
//     PlcTask Inputs/GVL_iXlinker.EtherCAT_Master_ATxxxx.Beckhoff_AT1xxx.Beckhoff_AT2xxxEK1122.A_0071_AT2050_0501_0023_AT2050_0501.A_0083_AT2050_5500_0016_AT2050_5500.FB_Inputs.Value_Channel[22] <-> FB Inputs/Value Channel 23
//     PlcTask Inputs/GVL_iXlinker.EtherCAT_Master_ATxxxx.Beckhoff_AT1xxx.Beckhoff_AT2xxxEK1122.A_0071_AT2050_0501_0023_AT2050_0501.A_0083_AT2050_5500_0016_AT2050_5500.FB_Inputs.Value_Channel[23] <-> FB Inputs/Value Channel 24
//     PlcTask Inputs/GVL_iXlinker.EtherCAT_Master_ATxxxx.Beckhoff_AT1xxx.Beckhoff_AT2xxxEK1122.A_0071_AT2050_0501_0023_AT2050_0501.A_0083_AT2050_5500_0016_AT2050_5500.FB_Inputs.Value_Channel[24] <-> FB Inputs/Value Channel 25
//     PlcTask Inputs/GVL_iXlinker.EtherCAT_Master_ATxxxx.Beckhoff_AT1xxx.Beckhoff_AT2xxxEK1122.A_0071_AT2050_0501_0023_AT2050_0501.A_0083_AT2050_5500_0016_AT2050_5500.FB_Inputs.Value_Channel[25] <-> FB Inputs/Value Channel 26
//     PlcTask Inputs/GVL_iXlinker.EtherCAT_Master_ATxxxx.Beckhoff_AT1xxx.Beckhoff_AT2xxxEK1122.A_0071_AT2050_0501_0023_AT2050_0501.A_0083_AT2050_5500_0016_AT2050_5500.FB_Inputs.Value_Channel[26] <-> FB Inputs/Value Channel 27
//     PlcTask Inputs/GVL_iXlinker.EtherCAT_Master_ATxxxx.Beckhoff_AT1xxx.Beckhoff_AT2xxxEK1122.A_0071_AT2050_0501_0023_AT2050_0501.A_0083_AT2050_5500_0016_AT2050_5500.FB_Inputs.Value_Channel[27] <-> FB Inputs/Value Channel 28
//     PlcTask Inputs/GVL_iXlinker.EtherCAT_Master_ATxxxx.Beckhoff_AT1xxx.Beckhoff_AT2xxxEK1122.A_0071_AT2050_0501_0023_AT2050_0501.A_0083_AT2050_5500_0016_AT2050_5500.FB_Inputs.Value_Channel[28] <-> FB Inputs/Value Channel 29
//     PlcTask Inputs/GVL_iXlinker.EtherCAT_Master_ATxxxx.Beckhoff_AT1xxx.Beckhoff_AT2xxxEK1122.A_0071_AT2050_0501_0023_AT2050_0501.A_0083_AT2050_5500_0016_AT2050_5500.FB_Inputs.Value_Channel[29] <-> FB Inputs/Value Channel 30
//     PlcTask Inputs/GVL_iXlinker.EtherCAT_Master_ATxxxx.Beckhoff_AT1xxx.Beckhoff_AT2xxxEK1122.A_0071_AT2050_0501_0023_AT2050_0501.A_0083_AT2050_5500_0016_AT2050_5500.FB_Inputs.Value_Channel[30] <-> FB Inputs/Value Channel 31
//     PlcTask Inputs/GVL_iXlinker.EtherCAT_Master_ATxxxx.Beckhoff_AT1xxx.Beckhoff_AT2xxxEK1122.A_0071_AT2050_0501_0023_AT2050_0501.A_0083_AT2050_5500_0016_AT2050_5500.FB_Inputs.Value_Channel[31] <-> FB Inputs/Value Channel 32
//     PlcTask Outputs/GVL_iXlinker.EtherCAT_Master_ATxxxx.Beckhoff_AT1xxx.Beckhoff_AT2xxxEK1122.A_0071_AT2050_0501_0023_AT2050_0501.A_0083_AT2050_5500_0016_AT2050_5500.FB_Outputs.Control <-> FB Outputs/Control
//     PlcTask Inputs/GVL_iXlinker.EtherCAT_Master_ATxxxx.Beckhoff_AT1xxx.Beckhoff_AT2xxxEK1122.A_0071_AT2050_0501_0023_AT2050_0501.A_0083_AT2050_5500_0016_AT2050_5500.WcState.WcState <-> WcState/WcState
//     PlcTask Inputs/GVL_iXlinker.EtherCAT_Master_ATxxxx.Beckhoff_AT1xxx.Beckhoff_AT2xxxEK1122.A_0071_AT2050_0501_0023_AT2050_0501.A_0083_AT2050_5500_0016_AT2050_5500.WcState.InputToggle <-> WcState/InputToggle
//     PlcTask Inputs/GVL_iXlinker.EtherCAT_Master_ATxxxx.Beckhoff_AT1xxx.Beckhoff_AT2xxxEK1122.A_0071_AT2050_0501_0023_AT2050_0501.A_0083_AT2050_5500_0016_AT2050_5500.InfoData.DcOutputShift <-> InfoData/DcOutputShift
//     PlcTask Inputs/GVL_iXlinker.EtherCAT_Master_ATxxxx.Beckhoff_AT1xxx.Beckhoff_AT2xxxEK1122.A_0071_AT2050_0501_0023_AT2050_0501.A_0083_AT2050_5500_0016_AT2050_5500.InfoData.DcInputShift <-> InfoData/DcInputShift
//     PlcTask Inputs/GVL_iXlinker.EtherCAT_Master_ATxxxx.Beckhoff_AT1xxx.Beckhoff_AT2xxxEK1122.A_0071_AT2050_0501_0023_AT2050_0501.A_0083_AT2050_5500_0016_AT2050_5500.InfoData.State <-> InfoData/State
//   PLC/PLC Instance <-> EtherCAT Master ATxxxx/Beckhoff AT1xxx/Beckhoff AT2xxxEK1122/A_0072(AT2050-0501-0024) (AT2050-0501)
//     PlcTask Inputs/GVL_iXlinker.EtherCAT_Master_ATxxxx.Beckhoff_AT1xxx.Beckhoff_AT2xxxEK1122.A_0072_AT2050_0501_0024_AT2050_0501.CC_Inputs.Status <-> CC Inputs/Status
//     PlcTask Inputs/GVL_iXlinker.EtherCAT_Master_ATxxxx.Beckhoff_AT1xxx.Beckhoff_AT2xxxEK1122.A_0072_AT2050_0501_0024_AT2050_0501.CC_Inputs.Current_actual_value_Ch[0] <-> CC Inputs/Current actual value Ch.1
//     PlcTask Inputs/GVL_iXlinker.EtherCAT_Master_ATxxxx.Beckhoff_AT1xxx.Beckhoff_AT2xxxEK1122.A_0072_AT2050_0501_0024_AT2050_0501.CC_Inputs.Current_actual_value_Ch[1] <-> CC Inputs/Current actual value Ch.2
//     PlcTask Inputs/GVL_iXlinker.EtherCAT_Master_ATxxxx.Beckhoff_AT1xxx.Beckhoff_AT2xxxEK1122.A_0072_AT2050_0501_0024_AT2050_0501.CC_Inputs.Current_actual_value_Ch[2] <-> CC Inputs/Current actual value Ch.3
//     PlcTask Inputs/GVL_iXlinker.EtherCAT_Master_ATxxxx.Beckhoff_AT1xxx.Beckhoff_AT2xxxEK1122.A_0072_AT2050_0501_0024_AT2050_0501.CC_Inputs.Current_actual_value_Ch[3] <-> CC Inputs/Current actual value Ch.4
//     PlcTask Inputs/GVL_iXlinker.EtherCAT_Master_ATxxxx.Beckhoff_AT1xxx.Beckhoff_AT2xxxEK1122.A_0072_AT2050_0501_0024_AT2050_0501.CC_Inputs.Current_actual_value_Ch[4] <-> CC Inputs/Current actual value Ch.5
//     PlcTask Inputs/GVL_iXlinker.EtherCAT_Master_ATxxxx.Beckhoff_AT1xxx.Beckhoff_AT2xxxEK1122.A_0072_AT2050_0501_0024_AT2050_0501.CC_Inputs.Current_actual_value_Ch[5] <-> CC Inputs/Current actual value Ch.6
//     PlcTask Inputs/GVL_iXlinker.EtherCAT_Master_ATxxxx.Beckhoff_AT1xxx.Beckhoff_AT2xxxEK1122.A_0072_AT2050_0501_0024_AT2050_0501.CC_Inputs.Current_actual_value_Ch[6] <-> CC Inputs/Current actual value Ch.7
//     PlcTask Inputs/GVL_iXlinker.EtherCAT_Master_ATxxxx.Beckhoff_AT1xxx.Beckhoff_AT2xxxEK1122.A_0072_AT2050_0501_0024_AT2050_0501.CC_Inputs.Current_actual_value_Ch[7] <-> CC Inputs/Current actual value Ch.8
//     PlcTask Inputs/GVL_iXlinker.EtherCAT_Master_ATxxxx.Beckhoff_AT1xxx.Beckhoff_AT2xxxEK1122.A_0072_AT2050_0501_0024_AT2050_0501.CC_Inputs.Current_actual_value_Ch[8] <-> CC Inputs/Current actual value Ch.9
//     PlcTask Inputs/GVL_iXlinker.EtherCAT_Master_ATxxxx.Beckhoff_AT1xxx.Beckhoff_AT2xxxEK1122.A_0072_AT2050_0501_0024_AT2050_0501.CC_Inputs.Current_actual_value_Ch[9] <-> CC Inputs/Current actual value Ch.10
//     PlcTask Inputs/GVL_iXlinker.EtherCAT_Master_ATxxxx.Beckhoff_AT1xxx.Beckhoff_AT2xxxEK1122.A_0072_AT2050_0501_0024_AT2050_0501.CC_Inputs.Current_actual_value_Ch[10] <-> CC Inputs/Current actual value Ch.11
//     PlcTask Inputs/GVL_iXlinker.EtherCAT_Master_ATxxxx.Beckhoff_AT1xxx.Beckhoff_AT2xxxEK1122.A_0072_AT2050_0501_0024_AT2050_0501.CC_Inputs.Current_actual_value_Ch[11] <-> CC Inputs/Current actual value Ch.12
//     PlcTask Inputs/GVL_iXlinker.EtherCAT_Master_ATxxxx.Beckhoff_AT1xxx.Beckhoff_AT2xxxEK1122.A_0072_AT2050_0501_0024_AT2050_0501.CC_Inputs.Current_actual_value_Ch[12] <-> CC Inputs/Current actual value Ch.13
//     PlcTask Inputs/GVL_iXlinker.EtherCAT_Master_ATxxxx.Beckhoff_AT1xxx.Beckhoff_AT2xxxEK1122.A_0072_AT2050_0501_0024_AT2050_0501.CC_Inputs.Current_actual_value_Ch[13] <-> CC Inputs/Current actual value Ch.14
//     PlcTask Inputs/GVL_iXlinker.EtherCAT_Master_ATxxxx.Beckhoff_AT1xxx.Beckhoff_AT2xxxEK1122.A_0072_AT2050_0501_0024_AT2050_0501.CC_Inputs.Current_actual_value_Ch[14] <-> CC Inputs/Current actual value Ch.15
//     PlcTask Outputs/GVL_iXlinker.EtherCAT_Master_ATxxxx.Beckhoff_AT1xxx.Beckhoff_AT2xxxEK1122.A_0072_AT2050_0501_0024_AT2050_0501.CC_Outputs.Control <-> CC Outputs/Control
//     PlcTask Outputs/GVL_iXlinker.EtherCAT_Master_ATxxxx.Beckhoff_AT1xxx.Beckhoff_AT2xxxEK1122.A_0072_AT2050_0501_0024_AT2050_0501.CC_Outputs.Current_setpoint_value_Ch[0] <-> CC Outputs/Current setpoint value Ch.1
//     PlcTask Outputs/GVL_iXlinker.EtherCAT_Master_ATxxxx.Beckhoff_AT1xxx.Beckhoff_AT2xxxEK1122.A_0072_AT2050_0501_0024_AT2050_0501.CC_Outputs.Current_setpoint_value_Ch[1] <-> CC Outputs/Current setpoint value Ch.2
//     PlcTask Outputs/GVL_iXlinker.EtherCAT_Master_ATxxxx.Beckhoff_AT1xxx.Beckhoff_AT2xxxEK1122.A_0072_AT2050_0501_0024_AT2050_0501.CC_Outputs.Current_setpoint_value_Ch[2] <-> CC Outputs/Current setpoint value Ch.3
//     PlcTask Outputs/GVL_iXlinker.EtherCAT_Master_ATxxxx.Beckhoff_AT1xxx.Beckhoff_AT2xxxEK1122.A_0072_AT2050_0501_0024_AT2050_0501.CC_Outputs.Current_setpoint_value_Ch[3] <-> CC Outputs/Current setpoint value Ch.4
//     PlcTask Outputs/GVL_iXlinker.EtherCAT_Master_ATxxxx.Beckhoff_AT1xxx.Beckhoff_AT2xxxEK1122.A_0072_AT2050_0501_0024_AT2050_0501.CC_Outputs.Current_setpoint_value_Ch[4] <-> CC Outputs/Current setpoint value Ch.5
//     PlcTask Outputs/GVL_iXlinker.EtherCAT_Master_ATxxxx.Beckhoff_AT1xxx.Beckhoff_AT2xxxEK1122.A_0072_AT2050_0501_0024_AT2050_0501.CC_Outputs.Current_setpoint_value_Ch[5] <-> CC Outputs/Current setpoint value Ch.6
//     PlcTask Outputs/GVL_iXlinker.EtherCAT_Master_ATxxxx.Beckhoff_AT1xxx.Beckhoff_AT2xxxEK1122.A_0072_AT2050_0501_0024_AT2050_0501.CC_Outputs.Current_setpoint_value_Ch[6] <-> CC Outputs/Current setpoint value Ch.7
//     PlcTask Outputs/GVL_iXlinker.EtherCAT_Master_ATxxxx.Beckhoff_AT1xxx.Beckhoff_AT2xxxEK1122.A_0072_AT2050_0501_0024_AT2050_0501.CC_Outputs.Current_setpoint_value_Ch[7] <-> CC Outputs/Current setpoint value Ch.8
//     PlcTask Outputs/GVL_iXlinker.EtherCAT_Master_ATxxxx.Beckhoff_AT1xxx.Beckhoff_AT2xxxEK1122.A_0072_AT2050_0501_0024_AT2050_0501.CC_Outputs.Current_setpoint_value_Ch[8] <-> CC Outputs/Current setpoint value Ch.9
//     PlcTask Outputs/GVL_iXlinker.EtherCAT_Master_ATxxxx.Beckhoff_AT1xxx.Beckhoff_AT2xxxEK1122.A_0072_AT2050_0501_0024_AT2050_0501.CC_Outputs.Current_setpoint_value_Ch[9] <-> CC Outputs/Current setpoint value Ch.10
//     PlcTask Outputs/GVL_iXlinker.EtherCAT_Master_ATxxxx.Beckhoff_AT1xxx.Beckhoff_AT2xxxEK1122.A_0072_AT2050_0501_0024_AT2050_0501.CC_Outputs.Current_setpoint_value_Ch[10] <-> CC Outputs/Current setpoint value Ch.11
//     PlcTask Outputs/GVL_iXlinker.EtherCAT_Master_ATxxxx.Beckhoff_AT1xxx.Beckhoff_AT2xxxEK1122.A_0072_AT2050_0501_0024_AT2050_0501.CC_Outputs.Current_setpoint_value_Ch[11] <-> CC Outputs/Current setpoint value Ch.12
//     PlcTask Outputs/GVL_iXlinker.EtherCAT_Master_ATxxxx.Beckhoff_AT1xxx.Beckhoff_AT2xxxEK1122.A_0072_AT2050_0501_0024_AT2050_0501.CC_Outputs.Current_setpoint_value_Ch[12] <-> CC Outputs/Current setpoint value Ch.13
//     PlcTask Outputs/GVL_iXlinker.EtherCAT_Master_ATxxxx.Beckhoff_AT1xxx.Beckhoff_AT2xxxEK1122.A_0072_AT2050_0501_0024_AT2050_0501.CC_Outputs.Current_setpoint_value_Ch[13] <-> CC Outputs/Current setpoint value Ch.14
//     PlcTask Outputs/GVL_iXlinker.EtherCAT_Master_ATxxxx.Beckhoff_AT1xxx.Beckhoff_AT2xxxEK1122.A_0072_AT2050_0501_0024_AT2050_0501.CC_Outputs.Current_setpoint_value_Ch[14] <-> CC Outputs/Current setpoint value Ch.15
//     PlcTask Inputs/GVL_iXlinker.EtherCAT_Master_ATxxxx.Beckhoff_AT1xxx.Beckhoff_AT2xxxEK1122.A_0072_AT2050_0501_0024_AT2050_0501.WcState.WcState <-> WcState/WcState
//     PlcTask Inputs/GVL_iXlinker.EtherCAT_Master_ATxxxx.Beckhoff_AT1xxx.Beckhoff_AT2xxxEK1122.A_0072_AT2050_0501_0024_AT2050_0501.WcState.InputToggle <-> WcState/InputToggle
//     PlcTask Inputs/GVL_iXlinker.EtherCAT_Master_ATxxxx.Beckhoff_AT1xxx.Beckhoff_AT2xxxEK1122.A_0072_AT2050_0501_0024_AT2050_0501.InfoData.AdsAddr <-> InfoData/AdsAddr
//     PlcTask Inputs/GVL_iXlinker.EtherCAT_Master_ATxxxx.Beckhoff_AT1xxx.Beckhoff_AT2xxxEK1122.A_0072_AT2050_0501_0024_AT2050_0501.InfoData.DcOutputShift <-> InfoData/DcOutputShift
//     PlcTask Inputs/GVL_iXlinker.EtherCAT_Master_ATxxxx.Beckhoff_AT1xxx.Beckhoff_AT2xxxEK1122.A_0072_AT2050_0501_0024_AT2050_0501.InfoData.DcInputShift <-> InfoData/DcInputShift
//     PlcTask Inputs/GVL_iXlinker.EtherCAT_Master_ATxxxx.Beckhoff_AT1xxx.Beckhoff_AT2xxxEK1122.A_0072_AT2050_0501_0024_AT2050_0501.InfoData.State <-> InfoData/State
//   PLC/PLC Instance <-> EtherCAT Master ATxxxx/Beckhoff AT1xxx/Beckhoff AT2xxxEK1122/A_0072(AT2050-0501-0024) (AT2050-0501)/A_0084(AT2050-5500-0017) (AT2050-5500)
//     PlcTask Inputs/GVL_iXlinker.EtherCAT_Master_ATxxxx.Beckhoff_AT1xxx.Beckhoff_AT2xxxEK1122.A_0072_AT2050_0501_0024_AT2050_0501.A_0084_AT2050_5500_0017_AT2050_5500.FB_Inputs.Status <-> FB Inputs/Status
//     PlcTask Inputs/GVL_iXlinker.EtherCAT_Master_ATxxxx.Beckhoff_AT1xxx.Beckhoff_AT2xxxEK1122.A_0072_AT2050_0501_0024_AT2050_0501.A_0084_AT2050_5500_0017_AT2050_5500.FB_Inputs.Value_Channel[0] <-> FB Inputs/Value Channel 01
//     PlcTask Inputs/GVL_iXlinker.EtherCAT_Master_ATxxxx.Beckhoff_AT1xxx.Beckhoff_AT2xxxEK1122.A_0072_AT2050_0501_0024_AT2050_0501.A_0084_AT2050_5500_0017_AT2050_5500.FB_Inputs.Value_Channel[1] <-> FB Inputs/Value Channel 02
//     PlcTask Inputs/GVL_iXlinker.EtherCAT_Master_ATxxxx.Beckhoff_AT1xxx.Beckhoff_AT2xxxEK1122.A_0072_AT2050_0501_0024_AT2050_0501.A_0084_AT2050_5500_0017_AT2050_5500.FB_Inputs.Value_Channel[2] <-> FB Inputs/Value Channel 03
//     PlcTask Inputs/GVL_iXlinker.EtherCAT_Master_ATxxxx.Beckhoff_AT1xxx.Beckhoff_AT2xxxEK1122.A_0072_AT2050_0501_0024_AT2050_0501.A_0084_AT2050_5500_0017_AT2050_5500.FB_Inputs.Value_Channel[3] <-> FB Inputs/Value Channel 04
//     PlcTask Inputs/GVL_iXlinker.EtherCAT_Master_ATxxxx.Beckhoff_AT1xxx.Beckhoff_AT2xxxEK1122.A_0072_AT2050_0501_0024_AT2050_0501.A_0084_AT2050_5500_0017_AT2050_5500.FB_Inputs.Value_Channel[4] <-> FB Inputs/Value Channel 05
//     PlcTask Inputs/GVL_iXlinker.EtherCAT_Master_ATxxxx.Beckhoff_AT1xxx.Beckhoff_AT2xxxEK1122.A_0072_AT2050_0501_0024_AT2050_0501.A_0084_AT2050_5500_0017_AT2050_5500.FB_Inputs.Value_Channel[5] <-> FB Inputs/Value Channel 06
//     PlcTask Inputs/GVL_iXlinker.EtherCAT_Master_ATxxxx.Beckhoff_AT1xxx.Beckhoff_AT2xxxEK1122.A_0072_AT2050_0501_0024_AT2050_0501.A_0084_AT2050_5500_0017_AT2050_5500.FB_Inputs.Value_Channel[6] <-> FB Inputs/Value Channel 07
//     PlcTask Inputs/GVL_iXlinker.EtherCAT_Master_ATxxxx.Beckhoff_AT1xxx.Beckhoff_AT2xxxEK1122.A_0072_AT2050_0501_0024_AT2050_0501.A_0084_AT2050_5500_0017_AT2050_5500.FB_Inputs.Value_Channel[7] <-> FB Inputs/Value Channel 08
//     PlcTask Inputs/GVL_iXlinker.EtherCAT_Master_ATxxxx.Beckhoff_AT1xxx.Beckhoff_AT2xxxEK1122.A_0072_AT2050_0501_0024_AT2050_0501.A_0084_AT2050_5500_0017_AT2050_5500.FB_Inputs.Value_Channel[8] <-> FB Inputs/Value Channel 09
//     PlcTask Inputs/GVL_iXlinker.EtherCAT_Master_ATxxxx.Beckhoff_AT1xxx.Beckhoff_AT2xxxEK1122.A_0072_AT2050_0501_0024_AT2050_0501.A_0084_AT2050_5500_0017_AT2050_5500.FB_Inputs.Value_Channel[9] <-> FB Inputs/Value Channel 10
//     PlcTask Inputs/GVL_iXlinker.EtherCAT_Master_ATxxxx.Beckhoff_AT1xxx.Beckhoff_AT2xxxEK1122.A_0072_AT2050_0501_0024_AT2050_0501.A_0084_AT2050_5500_0017_AT2050_5500.FB_Inputs.Value_Channel[10] <-> FB Inputs/Value Channel 11
//     PlcTask Inputs/GVL_iXlinker.EtherCAT_Master_ATxxxx.Beckhoff_AT1xxx.Beckhoff_AT2xxxEK1122.A_0072_AT2050_0501_0024_AT2050_0501.A_0084_AT2050_5500_0017_AT2050_5500.FB_Inputs.Value_Channel[11] <-> FB Inputs/Value Channel 12
//     PlcTask Inputs/GVL_iXlinker.EtherCAT_Master_ATxxxx.Beckhoff_AT1xxx.Beckhoff_AT2xxxEK1122.A_0072_AT2050_0501_0024_AT2050_0501.A_0084_AT2050_5500_0017_AT2050_5500.FB_Inputs.Value_Channel[12] <-> FB Inputs/Value Channel 13
//     PlcTask Inputs/GVL_iXlinker.EtherCAT_Master_ATxxxx.Beckhoff_AT1xxx.Beckhoff_AT2xxxEK1122.A_0072_AT2050_0501_0024_AT2050_0501.A_0084_AT2050_5500_0017_AT2050_5500.FB_Inputs.Value_Channel[13] <-> FB Inputs/Value Channel 14
//     PlcTask Inputs/GVL_iXlinker.EtherCAT_Master_ATxxxx.Beckhoff_AT1xxx.Beckhoff_AT2xxxEK1122.A_0072_AT2050_0501_0024_AT2050_0501.A_0084_AT2050_5500_0017_AT2050_5500.FB_Inputs.Value_Channel[14] <-> FB Inputs/Value Channel 15
//     PlcTask Inputs/GVL_iXlinker.EtherCAT_Master_ATxxxx.Beckhoff_AT1xxx.Beckhoff_AT2xxxEK1122.A_0072_AT2050_0501_0024_AT2050_0501.A_0084_AT2050_5500_0017_AT2050_5500.FB_Inputs.Value_Channel[15] <-> FB Inputs/Value Channel 16
//     PlcTask Inputs/GVL_iXlinker.EtherCAT_Master_ATxxxx.Beckhoff_AT1xxx.Beckhoff_AT2xxxEK1122.A_0072_AT2050_0501_0024_AT2050_0501.A_0084_AT2050_5500_0017_AT2050_5500.FB_Inputs.Value_Channel[16] <-> FB Inputs/Value Channel 17
//     PlcTask Inputs/GVL_iXlinker.EtherCAT_Master_ATxxxx.Beckhoff_AT1xxx.Beckhoff_AT2xxxEK1122.A_0072_AT2050_0501_0024_AT2050_0501.A_0084_AT2050_5500_0017_AT2050_5500.FB_Inputs.Value_Channel[17] <-> FB Inputs/Value Channel 18
//     PlcTask Inputs/GVL_iXlinker.EtherCAT_Master_ATxxxx.Beckhoff_AT1xxx.Beckhoff_AT2xxxEK1122.A_0072_AT2050_0501_0024_AT2050_0501.A_0084_AT2050_5500_0017_AT2050_5500.FB_Inputs.Value_Channel[18] <-> FB Inputs/Value Channel 19
//     PlcTask Inputs/GVL_iXlinker.EtherCAT_Master_ATxxxx.Beckhoff_AT1xxx.Beckhoff_AT2xxxEK1122.A_0072_AT2050_0501_0024_AT2050_0501.A_0084_AT2050_5500_0017_AT2050_5500.FB_Inputs.Value_Channel[19] <-> FB Inputs/Value Channel 20
//     PlcTask Inputs/GVL_iXlinker.EtherCAT_Master_ATxxxx.Beckhoff_AT1xxx.Beckhoff_AT2xxxEK1122.A_0072_AT2050_0501_0024_AT2050_0501.A_0084_AT2050_5500_0017_AT2050_5500.FB_Inputs.Value_Channel[20] <-> FB Inputs/Value Channel 21
//     PlcTask Inputs/GVL_iXlinker.EtherCAT_Master_ATxxxx.Beckhoff_AT1xxx.Beckhoff_AT2xxxEK1122.A_0072_AT2050_0501_0024_AT2050_0501.A_0084_AT2050_5500_0017_AT2050_5500.FB_Inputs.Value_Channel[21] <-> FB Inputs/Value Channel 22
//     PlcTask Inputs/GVL_iXlinker.EtherCAT_Master_ATxxxx.Beckhoff_AT1xxx.Beckhoff_AT2xxxEK1122.A_0072_AT2050_0501_0024_AT2050_0501.A_0084_AT2050_5500_0017_AT2050_5500.FB_Inputs.Value_Channel[22] <-> FB Inputs/Value Channel 23
//     PlcTask Inputs/GVL_iXlinker.EtherCAT_Master_ATxxxx.Beckhoff_AT1xxx.Beckhoff_AT2xxxEK1122.A_0072_AT2050_0501_0024_AT2050_0501.A_0084_AT2050_5500_0017_AT2050_5500.FB_Inputs.Value_Channel[23] <-> FB Inputs/Value Channel 24
//     PlcTask Inputs/GVL_iXlinker.EtherCAT_Master_ATxxxx.Beckhoff_AT1xxx.Beckhoff_AT2xxxEK1122.A_0072_AT2050_0501_0024_AT2050_0501.A_0084_AT2050_5500_0017_AT2050_5500.FB_Inputs.Value_Channel[24] <-> FB Inputs/Value Channel 25
//     PlcTask Inputs/GVL_iXlinker.EtherCAT_Master_ATxxxx.Beckhoff_AT1xxx.Beckhoff_AT2xxxEK1122.A_0072_AT2050_0501_0024_AT2050_0501.A_0084_AT2050_5500_0017_AT2050_5500.FB_Inputs.Value_Channel[25] <-> FB Inputs/Value Channel 26
//     PlcTask Inputs/GVL_iXlinker.EtherCAT_Master_ATxxxx.Beckhoff_AT1xxx.Beckhoff_AT2xxxEK1122.A_0072_AT2050_0501_0024_AT2050_0501.A_0084_AT2050_5500_0017_AT2050_5500.FB_Inputs.Value_Channel[26] <-> FB Inputs/Value Channel 27
//     PlcTask Inputs/GVL_iXlinker.EtherCAT_Master_ATxxxx.Beckhoff_AT1xxx.Beckhoff_AT2xxxEK1122.A_0072_AT2050_0501_0024_AT2050_0501.A_0084_AT2050_5500_0017_AT2050_5500.FB_Inputs.Value_Channel[27] <-> FB Inputs/Value Channel 28
//     PlcTask Inputs/GVL_iXlinker.EtherCAT_Master_ATxxxx.Beckhoff_AT1xxx.Beckhoff_AT2xxxEK1122.A_0072_AT2050_0501_0024_AT2050_0501.A_0084_AT2050_5500_0017_AT2050_5500.FB_Inputs.Value_Channel[28] <-> FB Inputs/Value Channel 29
//     PlcTask Inputs/GVL_iXlinker.EtherCAT_Master_ATxxxx.Beckhoff_AT1xxx.Beckhoff_AT2xxxEK1122.A_0072_AT2050_0501_0024_AT2050_0501.A_0084_AT2050_5500_0017_AT2050_5500.FB_Inputs.Value_Channel[29] <-> FB Inputs/Value Channel 30
//     PlcTask Inputs/GVL_iXlinker.EtherCAT_Master_ATxxxx.Beckhoff_AT1xxx.Beckhoff_AT2xxxEK1122.A_0072_AT2050_0501_0024_AT2050_0501.A_0084_AT2050_5500_0017_AT2050_5500.FB_Inputs.Value_Channel[30] <-> FB Inputs/Value Channel 31
//     PlcTask Inputs/GVL_iXlinker.EtherCAT_Master_ATxxxx.Beckhoff_AT1xxx.Beckhoff_AT2xxxEK1122.A_0072_AT2050_0501_0024_AT2050_0501.A_0084_AT2050_5500_0017_AT2050_5500.FB_Inputs.Value_Channel[31] <-> FB Inputs/Value Channel 32
//     PlcTask Outputs/GVL_iXlinker.EtherCAT_Master_ATxxxx.Beckhoff_AT1xxx.Beckhoff_AT2xxxEK1122.A_0072_AT2050_0501_0024_AT2050_0501.A_0084_AT2050_5500_0017_AT2050_5500.FB_Outputs.Control <-> FB Outputs/Control
//     PlcTask Inputs/GVL_iXlinker.EtherCAT_Master_ATxxxx.Beckhoff_AT1xxx.Beckhoff_AT2xxxEK1122.A_0072_AT2050_0501_0024_AT2050_0501.A_0084_AT2050_5500_0017_AT2050_5500.WcState.WcState <-> WcState/WcState
//     PlcTask Inputs/GVL_iXlinker.EtherCAT_Master_ATxxxx.Beckhoff_AT1xxx.Beckhoff_AT2xxxEK1122.A_0072_AT2050_0501_0024_AT2050_0501.A_0084_AT2050_5500_0017_AT2050_5500.WcState.InputToggle <-> WcState/InputToggle
//     PlcTask Inputs/GVL_iXlinker.EtherCAT_Master_ATxxxx.Beckhoff_AT1xxx.Beckhoff_AT2xxxEK1122.A_0072_AT2050_0501_0024_AT2050_0501.A_0084_AT2050_5500_0017_AT2050_5500.InfoData.DcOutputShift <-> InfoData/DcOutputShift
//     PlcTask Inputs/GVL_iXlinker.EtherCAT_Master_ATxxxx.Beckhoff_AT1xxx.Beckhoff_AT2xxxEK1122.A_0072_AT2050_0501_0024_AT2050_0501.A_0084_AT2050_5500_0017_AT2050_5500.InfoData.DcInputShift <-> InfoData/DcInputShift
//     PlcTask Inputs/GVL_iXlinker.EtherCAT_Master_ATxxxx.Beckhoff_AT1xxx.Beckhoff_AT2xxxEK1122.A_0072_AT2050_0501_0024_AT2050_0501.A_0084_AT2050_5500_0017_AT2050_5500.InfoData.State <-> InfoData/State
//   PLC/PLC Instance <-> EtherCAT Master ATxxxx/Beckhoff AT1xxx/A_0059(AT2000-5250-0018)
//     PlcTask Inputs/GVL_iXlinker.EtherCAT_Master_ATxxxx.Beckhoff_AT1xxx.A_0059_AT2000_5250_0018.FB_Inputs.Status <-> FB Inputs/Status
//     PlcTask Inputs/GVL_iXlinker.EtherCAT_Master_ATxxxx.Beckhoff_AT1xxx.A_0059_AT2000_5250_0018.FB_Inputs.Value_Channel[0] <-> FB Inputs/Value Channel 01
//     PlcTask Inputs/GVL_iXlinker.EtherCAT_Master_ATxxxx.Beckhoff_AT1xxx.A_0059_AT2000_5250_0018.FB_Inputs.Value_Channel[1] <-> FB Inputs/Value Channel 02
//     PlcTask Inputs/GVL_iXlinker.EtherCAT_Master_ATxxxx.Beckhoff_AT1xxx.A_0059_AT2000_5250_0018.FB_Inputs.Value_Channel[2] <-> FB Inputs/Value Channel 03
//     PlcTask Inputs/GVL_iXlinker.EtherCAT_Master_ATxxxx.Beckhoff_AT1xxx.A_0059_AT2000_5250_0018.FB_Inputs.Value_Channel[3] <-> FB Inputs/Value Channel 04
//     PlcTask Inputs/GVL_iXlinker.EtherCAT_Master_ATxxxx.Beckhoff_AT1xxx.A_0059_AT2000_5250_0018.FB_Inputs.Value_Channel[4] <-> FB Inputs/Value Channel 05
//     PlcTask Inputs/GVL_iXlinker.EtherCAT_Master_ATxxxx.Beckhoff_AT1xxx.A_0059_AT2000_5250_0018.FB_Inputs.Value_Channel[5] <-> FB Inputs/Value Channel 06
//     PlcTask Inputs/GVL_iXlinker.EtherCAT_Master_ATxxxx.Beckhoff_AT1xxx.A_0059_AT2000_5250_0018.FB_Inputs.Value_Channel[6] <-> FB Inputs/Value Channel 07
//     PlcTask Inputs/GVL_iXlinker.EtherCAT_Master_ATxxxx.Beckhoff_AT1xxx.A_0059_AT2000_5250_0018.FB_Inputs.Value_Channel[7] <-> FB Inputs/Value Channel 08
//     PlcTask Inputs/GVL_iXlinker.EtherCAT_Master_ATxxxx.Beckhoff_AT1xxx.A_0059_AT2000_5250_0018.FB_Inputs.Value_Channel[8] <-> FB Inputs/Value Channel 09
//     PlcTask Inputs/GVL_iXlinker.EtherCAT_Master_ATxxxx.Beckhoff_AT1xxx.A_0059_AT2000_5250_0018.FB_Inputs.Value_Channel[9] <-> FB Inputs/Value Channel 10
//     PlcTask Inputs/GVL_iXlinker.EtherCAT_Master_ATxxxx.Beckhoff_AT1xxx.A_0059_AT2000_5250_0018.FB_Inputs.Value_Channel[10] <-> FB Inputs/Value Channel 11
//     PlcTask Inputs/GVL_iXlinker.EtherCAT_Master_ATxxxx.Beckhoff_AT1xxx.A_0059_AT2000_5250_0018.FB_Inputs.Value_Channel[11] <-> FB Inputs/Value Channel 12
//     PlcTask Inputs/GVL_iXlinker.EtherCAT_Master_ATxxxx.Beckhoff_AT1xxx.A_0059_AT2000_5250_0018.FB_Inputs.Value_Channel[12] <-> FB Inputs/Value Channel 13
//     PlcTask Inputs/GVL_iXlinker.EtherCAT_Master_ATxxxx.Beckhoff_AT1xxx.A_0059_AT2000_5250_0018.FB_Inputs.Value_Channel[13] <-> FB Inputs/Value Channel 14
//     PlcTask Inputs/GVL_iXlinker.EtherCAT_Master_ATxxxx.Beckhoff_AT1xxx.A_0059_AT2000_5250_0018.FB_Inputs.Value_Channel[14] <-> FB Inputs/Value Channel 15
//     PlcTask Inputs/GVL_iXlinker.EtherCAT_Master_ATxxxx.Beckhoff_AT1xxx.A_0059_AT2000_5250_0018.FB_Inputs.Value_Channel[15] <-> FB Inputs/Value Channel 16
//     PlcTask Inputs/GVL_iXlinker.EtherCAT_Master_ATxxxx.Beckhoff_AT1xxx.A_0059_AT2000_5250_0018.FB_Inputs.Value_Channel[16] <-> FB Inputs/Value Channel 17
//     PlcTask Inputs/GVL_iXlinker.EtherCAT_Master_ATxxxx.Beckhoff_AT1xxx.A_0059_AT2000_5250_0018.FB_Inputs.Value_Channel[17] <-> FB Inputs/Value Channel 18
//     PlcTask Inputs/GVL_iXlinker.EtherCAT_Master_ATxxxx.Beckhoff_AT1xxx.A_0059_AT2000_5250_0018.FB_Inputs.Value_Channel[18] <-> FB Inputs/Value Channel 19
//     PlcTask Inputs/GVL_iXlinker.EtherCAT_Master_ATxxxx.Beckhoff_AT1xxx.A_0059_AT2000_5250_0018.FB_Inputs.Value_Channel[19] <-> FB Inputs/Value Channel 20
//     PlcTask Inputs/GVL_iXlinker.EtherCAT_Master_ATxxxx.Beckhoff_AT1xxx.A_0059_AT2000_5250_0018.FB_Inputs.Value_Channel[20] <-> FB Inputs/Value Channel 21
//     PlcTask Inputs/GVL_iXlinker.EtherCAT_Master_ATxxxx.Beckhoff_AT1xxx.A_0059_AT2000_5250_0018.FB_Inputs.Value_Channel[21] <-> FB Inputs/Value Channel 22
//     PlcTask Inputs/GVL_iXlinker.EtherCAT_Master_ATxxxx.Beckhoff_AT1xxx.A_0059_AT2000_5250_0018.FB_Inputs.Value_Channel[22] <-> FB Inputs/Value Channel 23
//     PlcTask Inputs/GVL_iXlinker.EtherCAT_Master_ATxxxx.Beckhoff_AT1xxx.A_0059_AT2000_5250_0018.FB_Inputs.Value_Channel[23] <-> FB Inputs/Value Channel 24
//     PlcTask Inputs/GVL_iXlinker.EtherCAT_Master_ATxxxx.Beckhoff_AT1xxx.A_0059_AT2000_5250_0018.FB_Inputs.Value_Channel[24] <-> FB Inputs/Value Channel 25
//     PlcTask Inputs/GVL_iXlinker.EtherCAT_Master_ATxxxx.Beckhoff_AT1xxx.A_0059_AT2000_5250_0018.FB_Inputs.Value_Channel[25] <-> FB Inputs/Value Channel 26
//     PlcTask Inputs/GVL_iXlinker.EtherCAT_Master_ATxxxx.Beckhoff_AT1xxx.A_0059_AT2000_5250_0018.FB_Inputs.Value_Channel[26] <-> FB Inputs/Value Channel 27
//     PlcTask Inputs/GVL_iXlinker.EtherCAT_Master_ATxxxx.Beckhoff_AT1xxx.A_0059_AT2000_5250_0018.FB_Inputs.Value_Channel[27] <-> FB Inputs/Value Channel 28
//     PlcTask Inputs/GVL_iXlinker.EtherCAT_Master_ATxxxx.Beckhoff_AT1xxx.A_0059_AT2000_5250_0018.FB_Inputs.Value_Channel[28] <-> FB Inputs/Value Channel 29
//     PlcTask Inputs/GVL_iXlinker.EtherCAT_Master_ATxxxx.Beckhoff_AT1xxx.A_0059_AT2000_5250_0018.FB_Inputs.Value_Channel[29] <-> FB Inputs/Value Channel 30
//     PlcTask Inputs/GVL_iXlinker.EtherCAT_Master_ATxxxx.Beckhoff_AT1xxx.A_0059_AT2000_5250_0018.FB_Inputs.Value_Channel[30] <-> FB Inputs/Value Channel 31
//     PlcTask Inputs/GVL_iXlinker.EtherCAT_Master_ATxxxx.Beckhoff_AT1xxx.A_0059_AT2000_5250_0018.FB_Inputs.Value_Channel[31] <-> FB Inputs/Value Channel 32
//     PlcTask Outputs/GVL_iXlinker.EtherCAT_Master_ATxxxx.Beckhoff_AT1xxx.A_0059_AT2000_5250_0018.FB_Outputs.Control <-> FB Outputs/Control
//     PlcTask Inputs/GVL_iXlinker.EtherCAT_Master_ATxxxx.Beckhoff_AT1xxx.A_0059_AT2000_5250_0018.WcState.WcState <-> WcState/WcState
//     PlcTask Inputs/GVL_iXlinker.EtherCAT_Master_ATxxxx.Beckhoff_AT1xxx.A_0059_AT2000_5250_0018.WcState.InputToggle <-> WcState/InputToggle
//     PlcTask Inputs/GVL_iXlinker.EtherCAT_Master_ATxxxx.Beckhoff_AT1xxx.A_0059_AT2000_5250_0018.InfoData.DcOutputShift <-> InfoData/DcOutputShift
//     PlcTask Inputs/GVL_iXlinker.EtherCAT_Master_ATxxxx.Beckhoff_AT1xxx.A_0059_AT2000_5250_0018.InfoData.DcInputShift <-> InfoData/DcInputShift
//     PlcTask Inputs/GVL_iXlinker.EtherCAT_Master_ATxxxx.Beckhoff_AT1xxx.A_0059_AT2000_5250_0018.InfoData.State <-> InfoData/State
//   PLC/PLC Instance <-> EtherCAT Master ATxxxx/Beckhoff ATH2xxx
//     PlcTask Inputs/GVL_iXlinker.EtherCAT_Master_ATxxxx.Beckhoff_ATH2xxx.InfoData.State <-> InfoData/State
//   PLC/PLC Instance <-> EtherCAT Master ATxxxx/Beckhoff ATH2xxx/Beckhoff ATH2xxxEK1122
//     PlcTask Inputs/GVL_iXlinker.EtherCAT_Master_ATxxxx.Beckhoff_ATH2xxx.Beckhoff_ATH2xxxEK1122.InfoData.State <-> InfoData/State
//   PLC/PLC Instance <-> EtherCAT Master ATxxxx/Beckhoff ATH2xxx/Beckhoff ATH2xxxEK1122/Beckhoff ATH2xxxsub EK1100
//     PlcTask Inputs/GVL_iXlinker.EtherCAT_Master_ATxxxx.Beckhoff_ATH2xxx.Beckhoff_ATH2xxxEK1122.Beckhoff_ATH2xxxsub_EK1100.InfoData.State <-> InfoData/State
//   PLC/PLC Instance <-> EtherCAT Master ATxxxx/Beckhoff ATH2xxx/Beckhoff ATH2xxxEK1122/A_0001(ATH2000-0250-0022)
//     PlcTask Inputs/GVL_iXlinker.EtherCAT_Master_ATxxxx.Beckhoff_ATH2xxx.Beckhoff_ATH2xxxEK1122.A_0001_ATH2000_0250_0022.CC_Inputs.Status <-> CC Inputs/Status
//     PlcTask Inputs/GVL_iXlinker.EtherCAT_Master_ATxxxx.Beckhoff_ATH2xxx.Beckhoff_ATH2xxxEK1122.A_0001_ATH2000_0250_0022.CC_Inputs.Current_actual_value_Ch[0] <-> CC Inputs/Current actual value Ch.1
//     PlcTask Inputs/GVL_iXlinker.EtherCAT_Master_ATxxxx.Beckhoff_ATH2xxx.Beckhoff_ATH2xxxEK1122.A_0001_ATH2000_0250_0022.CC_Inputs.Current_actual_value_Ch[1] <-> CC Inputs/Current actual value Ch.2
//     PlcTask Inputs/GVL_iXlinker.EtherCAT_Master_ATxxxx.Beckhoff_ATH2xxx.Beckhoff_ATH2xxxEK1122.A_0001_ATH2000_0250_0022.CC_Inputs.Current_actual_value_Ch[2] <-> CC Inputs/Current actual value Ch.3
//     PlcTask Inputs/GVL_iXlinker.EtherCAT_Master_ATxxxx.Beckhoff_ATH2xxx.Beckhoff_ATH2xxxEK1122.A_0001_ATH2000_0250_0022.CC_Inputs.Current_actual_value_Ch[3] <-> CC Inputs/Current actual value Ch.4
//     PlcTask Inputs/GVL_iXlinker.EtherCAT_Master_ATxxxx.Beckhoff_ATH2xxx.Beckhoff_ATH2xxxEK1122.A_0001_ATH2000_0250_0022.CC_Inputs.Current_actual_value_Ch[4] <-> CC Inputs/Current actual value Ch.5
//     PlcTask Inputs/GVL_iXlinker.EtherCAT_Master_ATxxxx.Beckhoff_ATH2xxx.Beckhoff_ATH2xxxEK1122.A_0001_ATH2000_0250_0022.CC_Inputs.Current_actual_value_Ch[5] <-> CC Inputs/Current actual value Ch.6
//     PlcTask Inputs/GVL_iXlinker.EtherCAT_Master_ATxxxx.Beckhoff_ATH2xxx.Beckhoff_ATH2xxxEK1122.A_0001_ATH2000_0250_0022.CC_Inputs.Current_actual_value_Ch[6] <-> CC Inputs/Current actual value Ch.7
//     PlcTask Inputs/GVL_iXlinker.EtherCAT_Master_ATxxxx.Beckhoff_ATH2xxx.Beckhoff_ATH2xxxEK1122.A_0001_ATH2000_0250_0022.CC_Inputs.Current_actual_value_Ch[7] <-> CC Inputs/Current actual value Ch.8
//     PlcTask Inputs/GVL_iXlinker.EtherCAT_Master_ATxxxx.Beckhoff_ATH2xxx.Beckhoff_ATH2xxxEK1122.A_0001_ATH2000_0250_0022.CC_Inputs.Current_actual_value_Ch[8] <-> CC Inputs/Current actual value Ch.9
//     PlcTask Inputs/GVL_iXlinker.EtherCAT_Master_ATxxxx.Beckhoff_ATH2xxx.Beckhoff_ATH2xxxEK1122.A_0001_ATH2000_0250_0022.CC_Inputs.Current_actual_value_Ch[9] <-> CC Inputs/Current actual value Ch.10
//     PlcTask Inputs/GVL_iXlinker.EtherCAT_Master_ATxxxx.Beckhoff_ATH2xxx.Beckhoff_ATH2xxxEK1122.A_0001_ATH2000_0250_0022.CC_Inputs.Current_actual_value_Ch[10] <-> CC Inputs/Current actual value Ch.11
//     PlcTask Inputs/GVL_iXlinker.EtherCAT_Master_ATxxxx.Beckhoff_ATH2xxx.Beckhoff_ATH2xxxEK1122.A_0001_ATH2000_0250_0022.CC_Inputs.Current_actual_value_Ch[11] <-> CC Inputs/Current actual value Ch.12
//     PlcTask Inputs/GVL_iXlinker.EtherCAT_Master_ATxxxx.Beckhoff_ATH2xxx.Beckhoff_ATH2xxxEK1122.A_0001_ATH2000_0250_0022.CC_Inputs.Current_actual_value_Ch[12] <-> CC Inputs/Current actual value Ch.13
//     PlcTask Inputs/GVL_iXlinker.EtherCAT_Master_ATxxxx.Beckhoff_ATH2xxx.Beckhoff_ATH2xxxEK1122.A_0001_ATH2000_0250_0022.CC_Inputs.Current_actual_value_Ch[13] <-> CC Inputs/Current actual value Ch.14
//     PlcTask Inputs/GVL_iXlinker.EtherCAT_Master_ATxxxx.Beckhoff_ATH2xxx.Beckhoff_ATH2xxxEK1122.A_0001_ATH2000_0250_0022.CC_Inputs.Current_actual_value_Ch[14] <-> CC Inputs/Current actual value Ch.15
//     PlcTask Outputs/GVL_iXlinker.EtherCAT_Master_ATxxxx.Beckhoff_ATH2xxx.Beckhoff_ATH2xxxEK1122.A_0001_ATH2000_0250_0022.CC_Outputs.Control <-> CC Outputs/Control
//     PlcTask Outputs/GVL_iXlinker.EtherCAT_Master_ATxxxx.Beckhoff_ATH2xxx.Beckhoff_ATH2xxxEK1122.A_0001_ATH2000_0250_0022.CC_Outputs.Current_setpoint_value_Ch[0] <-> CC Outputs/Current setpoint value Ch.1
//     PlcTask Outputs/GVL_iXlinker.EtherCAT_Master_ATxxxx.Beckhoff_ATH2xxx.Beckhoff_ATH2xxxEK1122.A_0001_ATH2000_0250_0022.CC_Outputs.Current_setpoint_value_Ch[1] <-> CC Outputs/Current setpoint value Ch.2
//     PlcTask Outputs/GVL_iXlinker.EtherCAT_Master_ATxxxx.Beckhoff_ATH2xxx.Beckhoff_ATH2xxxEK1122.A_0001_ATH2000_0250_0022.CC_Outputs.Current_setpoint_value_Ch[2] <-> CC Outputs/Current setpoint value Ch.3
//     PlcTask Outputs/GVL_iXlinker.EtherCAT_Master_ATxxxx.Beckhoff_ATH2xxx.Beckhoff_ATH2xxxEK1122.A_0001_ATH2000_0250_0022.CC_Outputs.Current_setpoint_value_Ch[3] <-> CC Outputs/Current setpoint value Ch.4
//     PlcTask Outputs/GVL_iXlinker.EtherCAT_Master_ATxxxx.Beckhoff_ATH2xxx.Beckhoff_ATH2xxxEK1122.A_0001_ATH2000_0250_0022.CC_Outputs.Current_setpoint_value_Ch[4] <-> CC Outputs/Current setpoint value Ch.5
//     PlcTask Outputs/GVL_iXlinker.EtherCAT_Master_ATxxxx.Beckhoff_ATH2xxx.Beckhoff_ATH2xxxEK1122.A_0001_ATH2000_0250_0022.CC_Outputs.Current_setpoint_value_Ch[5] <-> CC Outputs/Current setpoint value Ch.6
//     PlcTask Outputs/GVL_iXlinker.EtherCAT_Master_ATxxxx.Beckhoff_ATH2xxx.Beckhoff_ATH2xxxEK1122.A_0001_ATH2000_0250_0022.CC_Outputs.Current_setpoint_value_Ch[6] <-> CC Outputs/Current setpoint value Ch.7
//     PlcTask Outputs/GVL_iXlinker.EtherCAT_Master_ATxxxx.Beckhoff_ATH2xxx.Beckhoff_ATH2xxxEK1122.A_0001_ATH2000_0250_0022.CC_Outputs.Current_setpoint_value_Ch[7] <-> CC Outputs/Current setpoint value Ch.8
//     PlcTask Outputs/GVL_iXlinker.EtherCAT_Master_ATxxxx.Beckhoff_ATH2xxx.Beckhoff_ATH2xxxEK1122.A_0001_ATH2000_0250_0022.CC_Outputs.Current_setpoint_value_Ch[8] <-> CC Outputs/Current setpoint value Ch.9
//     PlcTask Outputs/GVL_iXlinker.EtherCAT_Master_ATxxxx.Beckhoff_ATH2xxx.Beckhoff_ATH2xxxEK1122.A_0001_ATH2000_0250_0022.CC_Outputs.Current_setpoint_value_Ch[9] <-> CC Outputs/Current setpoint value Ch.10
//     PlcTask Outputs/GVL_iXlinker.EtherCAT_Master_ATxxxx.Beckhoff_ATH2xxx.Beckhoff_ATH2xxxEK1122.A_0001_ATH2000_0250_0022.CC_Outputs.Current_setpoint_value_Ch[10] <-> CC Outputs/Current setpoint value Ch.11
//     PlcTask Outputs/GVL_iXlinker.EtherCAT_Master_ATxxxx.Beckhoff_ATH2xxx.Beckhoff_ATH2xxxEK1122.A_0001_ATH2000_0250_0022.CC_Outputs.Current_setpoint_value_Ch[11] <-> CC Outputs/Current setpoint value Ch.12
//     PlcTask Outputs/GVL_iXlinker.EtherCAT_Master_ATxxxx.Beckhoff_ATH2xxx.Beckhoff_ATH2xxxEK1122.A_0001_ATH2000_0250_0022.CC_Outputs.Current_setpoint_value_Ch[12] <-> CC Outputs/Current setpoint value Ch.13
//     PlcTask Outputs/GVL_iXlinker.EtherCAT_Master_ATxxxx.Beckhoff_ATH2xxx.Beckhoff_ATH2xxxEK1122.A_0001_ATH2000_0250_0022.CC_Outputs.Current_setpoint_value_Ch[13] <-> CC Outputs/Current setpoint value Ch.14
//     PlcTask Outputs/GVL_iXlinker.EtherCAT_Master_ATxxxx.Beckhoff_ATH2xxx.Beckhoff_ATH2xxxEK1122.A_0001_ATH2000_0250_0022.CC_Outputs.Current_setpoint_value_Ch[14] <-> CC Outputs/Current setpoint value Ch.15
//     PlcTask Inputs/GVL_iXlinker.EtherCAT_Master_ATxxxx.Beckhoff_ATH2xxx.Beckhoff_ATH2xxxEK1122.A_0001_ATH2000_0250_0022.WcState.WcState <-> WcState/WcState
//     PlcTask Inputs/GVL_iXlinker.EtherCAT_Master_ATxxxx.Beckhoff_ATH2xxx.Beckhoff_ATH2xxxEK1122.A_0001_ATH2000_0250_0022.WcState.InputToggle <-> WcState/InputToggle
//     PlcTask Inputs/GVL_iXlinker.EtherCAT_Master_ATxxxx.Beckhoff_ATH2xxx.Beckhoff_ATH2xxxEK1122.A_0001_ATH2000_0250_0022.InfoData.AdsAddr <-> InfoData/AdsAddr
//     PlcTask Inputs/GVL_iXlinker.EtherCAT_Master_ATxxxx.Beckhoff_ATH2xxx.Beckhoff_ATH2xxxEK1122.A_0001_ATH2000_0250_0022.InfoData.DcOutputShift <-> InfoData/DcOutputShift
//     PlcTask Inputs/GVL_iXlinker.EtherCAT_Master_ATxxxx.Beckhoff_ATH2xxx.Beckhoff_ATH2xxxEK1122.A_0001_ATH2000_0250_0022.InfoData.DcInputShift <-> InfoData/DcInputShift
//     PlcTask Inputs/GVL_iXlinker.EtherCAT_Master_ATxxxx.Beckhoff_ATH2xxx.Beckhoff_ATH2xxxEK1122.A_0001_ATH2000_0250_0022.InfoData.State <-> InfoData/State
//   PLC/PLC Instance <-> EtherCAT Master ATxxxx/Beckhoff ATH2xxx/Beckhoff ATH2xxxEK1122/A_0001(ATH2000-0250-0022)/A_0014(ATH2050-5501-0022)
//     PlcTask Inputs/GVL_iXlinker.EtherCAT_Master_ATxxxx.Beckhoff_ATH2xxx.Beckhoff_ATH2xxxEK1122.A_0001_ATH2000_0250_0022.A_0014_ATH2050_5501_0022.FB_Inputs.BinaryData <-> FB Inputs/BinaryData
//     PlcTask Outputs/GVL_iXlinker.EtherCAT_Master_ATxxxx.Beckhoff_ATH2xxx.Beckhoff_ATH2xxxEK1122.A_0001_ATH2000_0250_0022.A_0014_ATH2050_5501_0022.FB_Outputs.Control <-> FB Outputs/Control
//     PlcTask Inputs/GVL_iXlinker.EtherCAT_Master_ATxxxx.Beckhoff_ATH2xxx.Beckhoff_ATH2xxxEK1122.A_0001_ATH2000_0250_0022.A_0014_ATH2050_5501_0022.WcState.WcState <-> WcState/WcState
//     PlcTask Inputs/GVL_iXlinker.EtherCAT_Master_ATxxxx.Beckhoff_ATH2xxx.Beckhoff_ATH2xxxEK1122.A_0001_ATH2000_0250_0022.A_0014_ATH2050_5501_0022.WcState.InputToggle <-> WcState/InputToggle
//     PlcTask Inputs/GVL_iXlinker.EtherCAT_Master_ATxxxx.Beckhoff_ATH2xxx.Beckhoff_ATH2xxxEK1122.A_0001_ATH2000_0250_0022.A_0014_ATH2050_5501_0022.InfoData.DcOutputShift <-> InfoData/DcOutputShift
//     PlcTask Inputs/GVL_iXlinker.EtherCAT_Master_ATxxxx.Beckhoff_ATH2xxx.Beckhoff_ATH2xxxEK1122.A_0001_ATH2000_0250_0022.A_0014_ATH2050_5501_0022.InfoData.DcInputShift <-> InfoData/DcInputShift
//     PlcTask Inputs/GVL_iXlinker.EtherCAT_Master_ATxxxx.Beckhoff_ATH2xxx.Beckhoff_ATH2xxxEK1122.A_0001_ATH2000_0250_0022.A_0014_ATH2050_5501_0022.InfoData.State <-> InfoData/State
//   PLC/PLC Instance <-> EtherCAT Master ATxxxx/Beckhoff ATH2xxx/Beckhoff ATH2xxxEK1122/A_0002(ATH2000-0250-0023)
//     PlcTask Inputs/GVL_iXlinker.EtherCAT_Master_ATxxxx.Beckhoff_ATH2xxx.Beckhoff_ATH2xxxEK1122.A_0002_ATH2000_0250_0023.CC_Inputs.Status <-> CC Inputs/Status
//     PlcTask Inputs/GVL_iXlinker.EtherCAT_Master_ATxxxx.Beckhoff_ATH2xxx.Beckhoff_ATH2xxxEK1122.A_0002_ATH2000_0250_0023.CC_Inputs.Current_actual_value_Ch[0] <-> CC Inputs/Current actual value Ch.1
//     PlcTask Inputs/GVL_iXlinker.EtherCAT_Master_ATxxxx.Beckhoff_ATH2xxx.Beckhoff_ATH2xxxEK1122.A_0002_ATH2000_0250_0023.CC_Inputs.Current_actual_value_Ch[1] <-> CC Inputs/Current actual value Ch.2
//     PlcTask Inputs/GVL_iXlinker.EtherCAT_Master_ATxxxx.Beckhoff_ATH2xxx.Beckhoff_ATH2xxxEK1122.A_0002_ATH2000_0250_0023.CC_Inputs.Current_actual_value_Ch[2] <-> CC Inputs/Current actual value Ch.3
//     PlcTask Inputs/GVL_iXlinker.EtherCAT_Master_ATxxxx.Beckhoff_ATH2xxx.Beckhoff_ATH2xxxEK1122.A_0002_ATH2000_0250_0023.CC_Inputs.Current_actual_value_Ch[3] <-> CC Inputs/Current actual value Ch.4
//     PlcTask Inputs/GVL_iXlinker.EtherCAT_Master_ATxxxx.Beckhoff_ATH2xxx.Beckhoff_ATH2xxxEK1122.A_0002_ATH2000_0250_0023.CC_Inputs.Current_actual_value_Ch[4] <-> CC Inputs/Current actual value Ch.5
//     PlcTask Inputs/GVL_iXlinker.EtherCAT_Master_ATxxxx.Beckhoff_ATH2xxx.Beckhoff_ATH2xxxEK1122.A_0002_ATH2000_0250_0023.CC_Inputs.Current_actual_value_Ch[5] <-> CC Inputs/Current actual value Ch.6
//     PlcTask Inputs/GVL_iXlinker.EtherCAT_Master_ATxxxx.Beckhoff_ATH2xxx.Beckhoff_ATH2xxxEK1122.A_0002_ATH2000_0250_0023.CC_Inputs.Current_actual_value_Ch[6] <-> CC Inputs/Current actual value Ch.7
//     PlcTask Inputs/GVL_iXlinker.EtherCAT_Master_ATxxxx.Beckhoff_ATH2xxx.Beckhoff_ATH2xxxEK1122.A_0002_ATH2000_0250_0023.CC_Inputs.Current_actual_value_Ch[7] <-> CC Inputs/Current actual value Ch.8
//     PlcTask Inputs/GVL_iXlinker.EtherCAT_Master_ATxxxx.Beckhoff_ATH2xxx.Beckhoff_ATH2xxxEK1122.A_0002_ATH2000_0250_0023.CC_Inputs.Current_actual_value_Ch[8] <-> CC Inputs/Current actual value Ch.9
//     PlcTask Inputs/GVL_iXlinker.EtherCAT_Master_ATxxxx.Beckhoff_ATH2xxx.Beckhoff_ATH2xxxEK1122.A_0002_ATH2000_0250_0023.CC_Inputs.Current_actual_value_Ch[9] <-> CC Inputs/Current actual value Ch.10
//     PlcTask Inputs/GVL_iXlinker.EtherCAT_Master_ATxxxx.Beckhoff_ATH2xxx.Beckhoff_ATH2xxxEK1122.A_0002_ATH2000_0250_0023.CC_Inputs.Current_actual_value_Ch[10] <-> CC Inputs/Current actual value Ch.11
//     PlcTask Inputs/GVL_iXlinker.EtherCAT_Master_ATxxxx.Beckhoff_ATH2xxx.Beckhoff_ATH2xxxEK1122.A_0002_ATH2000_0250_0023.CC_Inputs.Current_actual_value_Ch[11] <-> CC Inputs/Current actual value Ch.12
//     PlcTask Inputs/GVL_iXlinker.EtherCAT_Master_ATxxxx.Beckhoff_ATH2xxx.Beckhoff_ATH2xxxEK1122.A_0002_ATH2000_0250_0023.CC_Inputs.Current_actual_value_Ch[12] <-> CC Inputs/Current actual value Ch.13
//     PlcTask Inputs/GVL_iXlinker.EtherCAT_Master_ATxxxx.Beckhoff_ATH2xxx.Beckhoff_ATH2xxxEK1122.A_0002_ATH2000_0250_0023.CC_Inputs.Current_actual_value_Ch[13] <-> CC Inputs/Current actual value Ch.14
//     PlcTask Inputs/GVL_iXlinker.EtherCAT_Master_ATxxxx.Beckhoff_ATH2xxx.Beckhoff_ATH2xxxEK1122.A_0002_ATH2000_0250_0023.CC_Inputs.Current_actual_value_Ch[14] <-> CC Inputs/Current actual value Ch.15
//     PlcTask Outputs/GVL_iXlinker.EtherCAT_Master_ATxxxx.Beckhoff_ATH2xxx.Beckhoff_ATH2xxxEK1122.A_0002_ATH2000_0250_0023.CC_Outputs.Control <-> CC Outputs/Control
//     PlcTask Outputs/GVL_iXlinker.EtherCAT_Master_ATxxxx.Beckhoff_ATH2xxx.Beckhoff_ATH2xxxEK1122.A_0002_ATH2000_0250_0023.CC_Outputs.Current_setpoint_value_Ch[0] <-> CC Outputs/Current setpoint value Ch.1
//     PlcTask Outputs/GVL_iXlinker.EtherCAT_Master_ATxxxx.Beckhoff_ATH2xxx.Beckhoff_ATH2xxxEK1122.A_0002_ATH2000_0250_0023.CC_Outputs.Current_setpoint_value_Ch[1] <-> CC Outputs/Current setpoint value Ch.2
//     PlcTask Outputs/GVL_iXlinker.EtherCAT_Master_ATxxxx.Beckhoff_ATH2xxx.Beckhoff_ATH2xxxEK1122.A_0002_ATH2000_0250_0023.CC_Outputs.Current_setpoint_value_Ch[2] <-> CC Outputs/Current setpoint value Ch.3
//     PlcTask Outputs/GVL_iXlinker.EtherCAT_Master_ATxxxx.Beckhoff_ATH2xxx.Beckhoff_ATH2xxxEK1122.A_0002_ATH2000_0250_0023.CC_Outputs.Current_setpoint_value_Ch[3] <-> CC Outputs/Current setpoint value Ch.4
//     PlcTask Outputs/GVL_iXlinker.EtherCAT_Master_ATxxxx.Beckhoff_ATH2xxx.Beckhoff_ATH2xxxEK1122.A_0002_ATH2000_0250_0023.CC_Outputs.Current_setpoint_value_Ch[4] <-> CC Outputs/Current setpoint value Ch.5
//     PlcTask Outputs/GVL_iXlinker.EtherCAT_Master_ATxxxx.Beckhoff_ATH2xxx.Beckhoff_ATH2xxxEK1122.A_0002_ATH2000_0250_0023.CC_Outputs.Current_setpoint_value_Ch[5] <-> CC Outputs/Current setpoint value Ch.6
//     PlcTask Outputs/GVL_iXlinker.EtherCAT_Master_ATxxxx.Beckhoff_ATH2xxx.Beckhoff_ATH2xxxEK1122.A_0002_ATH2000_0250_0023.CC_Outputs.Current_setpoint_value_Ch[6] <-> CC Outputs/Current setpoint value Ch.7
//     PlcTask Outputs/GVL_iXlinker.EtherCAT_Master_ATxxxx.Beckhoff_ATH2xxx.Beckhoff_ATH2xxxEK1122.A_0002_ATH2000_0250_0023.CC_Outputs.Current_setpoint_value_Ch[7] <-> CC Outputs/Current setpoint value Ch.8
//     PlcTask Outputs/GVL_iXlinker.EtherCAT_Master_ATxxxx.Beckhoff_ATH2xxx.Beckhoff_ATH2xxxEK1122.A_0002_ATH2000_0250_0023.CC_Outputs.Current_setpoint_value_Ch[8] <-> CC Outputs/Current setpoint value Ch.9
//     PlcTask Outputs/GVL_iXlinker.EtherCAT_Master_ATxxxx.Beckhoff_ATH2xxx.Beckhoff_ATH2xxxEK1122.A_0002_ATH2000_0250_0023.CC_Outputs.Current_setpoint_value_Ch[9] <-> CC Outputs/Current setpoint value Ch.10
//     PlcTask Outputs/GVL_iXlinker.EtherCAT_Master_ATxxxx.Beckhoff_ATH2xxx.Beckhoff_ATH2xxxEK1122.A_0002_ATH2000_0250_0023.CC_Outputs.Current_setpoint_value_Ch[10] <-> CC Outputs/Current setpoint value Ch.11
//     PlcTask Outputs/GVL_iXlinker.EtherCAT_Master_ATxxxx.Beckhoff_ATH2xxx.Beckhoff_ATH2xxxEK1122.A_0002_ATH2000_0250_0023.CC_Outputs.Current_setpoint_value_Ch[11] <-> CC Outputs/Current setpoint value Ch.12
//     PlcTask Outputs/GVL_iXlinker.EtherCAT_Master_ATxxxx.Beckhoff_ATH2xxx.Beckhoff_ATH2xxxEK1122.A_0002_ATH2000_0250_0023.CC_Outputs.Current_setpoint_value_Ch[12] <-> CC Outputs/Current setpoint value Ch.13
//     PlcTask Outputs/GVL_iXlinker.EtherCAT_Master_ATxxxx.Beckhoff_ATH2xxx.Beckhoff_ATH2xxxEK1122.A_0002_ATH2000_0250_0023.CC_Outputs.Current_setpoint_value_Ch[13] <-> CC Outputs/Current setpoint value Ch.14
//     PlcTask Outputs/GVL_iXlinker.EtherCAT_Master_ATxxxx.Beckhoff_ATH2xxx.Beckhoff_ATH2xxxEK1122.A_0002_ATH2000_0250_0023.CC_Outputs.Current_setpoint_value_Ch[14] <-> CC Outputs/Current setpoint value Ch.15
//     PlcTask Inputs/GVL_iXlinker.EtherCAT_Master_ATxxxx.Beckhoff_ATH2xxx.Beckhoff_ATH2xxxEK1122.A_0002_ATH2000_0250_0023.WcState.WcState <-> WcState/WcState
//     PlcTask Inputs/GVL_iXlinker.EtherCAT_Master_ATxxxx.Beckhoff_ATH2xxx.Beckhoff_ATH2xxxEK1122.A_0002_ATH2000_0250_0023.WcState.InputToggle <-> WcState/InputToggle
//     PlcTask Inputs/GVL_iXlinker.EtherCAT_Master_ATxxxx.Beckhoff_ATH2xxx.Beckhoff_ATH2xxxEK1122.A_0002_ATH2000_0250_0023.InfoData.AdsAddr <-> InfoData/AdsAddr
//     PlcTask Inputs/GVL_iXlinker.EtherCAT_Master_ATxxxx.Beckhoff_ATH2xxx.Beckhoff_ATH2xxxEK1122.A_0002_ATH2000_0250_0023.InfoData.DcOutputShift <-> InfoData/DcOutputShift
//     PlcTask Inputs/GVL_iXlinker.EtherCAT_Master_ATxxxx.Beckhoff_ATH2xxx.Beckhoff_ATH2xxxEK1122.A_0002_ATH2000_0250_0023.InfoData.DcInputShift <-> InfoData/DcInputShift
//     PlcTask Inputs/GVL_iXlinker.EtherCAT_Master_ATxxxx.Beckhoff_ATH2xxx.Beckhoff_ATH2xxxEK1122.A_0002_ATH2000_0250_0023.InfoData.State <-> InfoData/State
//   PLC/PLC Instance <-> EtherCAT Master ATxxxx/Beckhoff ATH2xxx/Beckhoff ATH2xxxEK1122/A_0002(ATH2000-0250-0023)/A_0015(ATH2040-5250-0022)
//     PlcTask Inputs/GVL_iXlinker.EtherCAT_Master_ATxxxx.Beckhoff_ATH2xxx.Beckhoff_ATH2xxxEK1122.A_0002_ATH2000_0250_0023.A_0015_ATH2040_5250_0022.FB_Inputs.BinaryData <-> FB Inputs/BinaryData
//     PlcTask Outputs/GVL_iXlinker.EtherCAT_Master_ATxxxx.Beckhoff_ATH2xxx.Beckhoff_ATH2xxxEK1122.A_0002_ATH2000_0250_0023.A_0015_ATH2040_5250_0022.FB_Outputs.Control <-> FB Outputs/Control
//     PlcTask Inputs/GVL_iXlinker.EtherCAT_Master_ATxxxx.Beckhoff_ATH2xxx.Beckhoff_ATH2xxxEK1122.A_0002_ATH2000_0250_0023.A_0015_ATH2040_5250_0022.WcState.WcState <-> WcState/WcState
//     PlcTask Inputs/GVL_iXlinker.EtherCAT_Master_ATxxxx.Beckhoff_ATH2xxx.Beckhoff_ATH2xxxEK1122.A_0002_ATH2000_0250_0023.A_0015_ATH2040_5250_0022.WcState.InputToggle <-> WcState/InputToggle
//     PlcTask Inputs/GVL_iXlinker.EtherCAT_Master_ATxxxx.Beckhoff_ATH2xxx.Beckhoff_ATH2xxxEK1122.A_0002_ATH2000_0250_0023.A_0015_ATH2040_5250_0022.InfoData.DcOutputShift <-> InfoData/DcOutputShift
//     PlcTask Inputs/GVL_iXlinker.EtherCAT_Master_ATxxxx.Beckhoff_ATH2xxx.Beckhoff_ATH2xxxEK1122.A_0002_ATH2000_0250_0023.A_0015_ATH2040_5250_0022.InfoData.DcInputShift <-> InfoData/DcInputShift
//     PlcTask Inputs/GVL_iXlinker.EtherCAT_Master_ATxxxx.Beckhoff_ATH2xxx.Beckhoff_ATH2xxxEK1122.A_0002_ATH2000_0250_0023.A_0015_ATH2040_5250_0022.InfoData.State <-> InfoData/State
//   PLC/PLC Instance <-> EtherCAT Master ATxxxx/Beckhoff ATH2xxx/Beckhoff ATH2xxxEK1122/A_0003(ATH2000-0250-0024)
//     PlcTask Inputs/GVL_iXlinker.EtherCAT_Master_ATxxxx.Beckhoff_ATH2xxx.Beckhoff_ATH2xxxEK1122.A_0003_ATH2000_0250_0024.CC_Inputs.Status <-> CC Inputs/Status
//     PlcTask Inputs/GVL_iXlinker.EtherCAT_Master_ATxxxx.Beckhoff_ATH2xxx.Beckhoff_ATH2xxxEK1122.A_0003_ATH2000_0250_0024.CC_Inputs.Current_actual_value_Ch[0] <-> CC Inputs/Current actual value Ch.1
//     PlcTask Inputs/GVL_iXlinker.EtherCAT_Master_ATxxxx.Beckhoff_ATH2xxx.Beckhoff_ATH2xxxEK1122.A_0003_ATH2000_0250_0024.CC_Inputs.Current_actual_value_Ch[1] <-> CC Inputs/Current actual value Ch.2
//     PlcTask Inputs/GVL_iXlinker.EtherCAT_Master_ATxxxx.Beckhoff_ATH2xxx.Beckhoff_ATH2xxxEK1122.A_0003_ATH2000_0250_0024.CC_Inputs.Current_actual_value_Ch[2] <-> CC Inputs/Current actual value Ch.3
//     PlcTask Inputs/GVL_iXlinker.EtherCAT_Master_ATxxxx.Beckhoff_ATH2xxx.Beckhoff_ATH2xxxEK1122.A_0003_ATH2000_0250_0024.CC_Inputs.Current_actual_value_Ch[3] <-> CC Inputs/Current actual value Ch.4
//     PlcTask Inputs/GVL_iXlinker.EtherCAT_Master_ATxxxx.Beckhoff_ATH2xxx.Beckhoff_ATH2xxxEK1122.A_0003_ATH2000_0250_0024.CC_Inputs.Current_actual_value_Ch[4] <-> CC Inputs/Current actual value Ch.5
//     PlcTask Inputs/GVL_iXlinker.EtherCAT_Master_ATxxxx.Beckhoff_ATH2xxx.Beckhoff_ATH2xxxEK1122.A_0003_ATH2000_0250_0024.CC_Inputs.Current_actual_value_Ch[5] <-> CC Inputs/Current actual value Ch.6
//     PlcTask Inputs/GVL_iXlinker.EtherCAT_Master_ATxxxx.Beckhoff_ATH2xxx.Beckhoff_ATH2xxxEK1122.A_0003_ATH2000_0250_0024.CC_Inputs.Current_actual_value_Ch[6] <-> CC Inputs/Current actual value Ch.7
//     PlcTask Inputs/GVL_iXlinker.EtherCAT_Master_ATxxxx.Beckhoff_ATH2xxx.Beckhoff_ATH2xxxEK1122.A_0003_ATH2000_0250_0024.CC_Inputs.Current_actual_value_Ch[7] <-> CC Inputs/Current actual value Ch.8
//     PlcTask Inputs/GVL_iXlinker.EtherCAT_Master_ATxxxx.Beckhoff_ATH2xxx.Beckhoff_ATH2xxxEK1122.A_0003_ATH2000_0250_0024.CC_Inputs.Current_actual_value_Ch[8] <-> CC Inputs/Current actual value Ch.9
//     PlcTask Inputs/GVL_iXlinker.EtherCAT_Master_ATxxxx.Beckhoff_ATH2xxx.Beckhoff_ATH2xxxEK1122.A_0003_ATH2000_0250_0024.CC_Inputs.Current_actual_value_Ch[9] <-> CC Inputs/Current actual value Ch.10
//     PlcTask Inputs/GVL_iXlinker.EtherCAT_Master_ATxxxx.Beckhoff_ATH2xxx.Beckhoff_ATH2xxxEK1122.A_0003_ATH2000_0250_0024.CC_Inputs.Current_actual_value_Ch[10] <-> CC Inputs/Current actual value Ch.11
//     PlcTask Inputs/GVL_iXlinker.EtherCAT_Master_ATxxxx.Beckhoff_ATH2xxx.Beckhoff_ATH2xxxEK1122.A_0003_ATH2000_0250_0024.CC_Inputs.Current_actual_value_Ch[11] <-> CC Inputs/Current actual value Ch.12
//     PlcTask Inputs/GVL_iXlinker.EtherCAT_Master_ATxxxx.Beckhoff_ATH2xxx.Beckhoff_ATH2xxxEK1122.A_0003_ATH2000_0250_0024.CC_Inputs.Current_actual_value_Ch[12] <-> CC Inputs/Current actual value Ch.13
//     PlcTask Inputs/GVL_iXlinker.EtherCAT_Master_ATxxxx.Beckhoff_ATH2xxx.Beckhoff_ATH2xxxEK1122.A_0003_ATH2000_0250_0024.CC_Inputs.Current_actual_value_Ch[13] <-> CC Inputs/Current actual value Ch.14
//     PlcTask Inputs/GVL_iXlinker.EtherCAT_Master_ATxxxx.Beckhoff_ATH2xxx.Beckhoff_ATH2xxxEK1122.A_0003_ATH2000_0250_0024.CC_Inputs.Current_actual_value_Ch[14] <-> CC Inputs/Current actual value Ch.15
//     PlcTask Outputs/GVL_iXlinker.EtherCAT_Master_ATxxxx.Beckhoff_ATH2xxx.Beckhoff_ATH2xxxEK1122.A_0003_ATH2000_0250_0024.CC_Outputs.Control <-> CC Outputs/Control
//     PlcTask Outputs/GVL_iXlinker.EtherCAT_Master_ATxxxx.Beckhoff_ATH2xxx.Beckhoff_ATH2xxxEK1122.A_0003_ATH2000_0250_0024.CC_Outputs.Current_setpoint_value_Ch[0] <-> CC Outputs/Current setpoint value Ch.1
//     PlcTask Outputs/GVL_iXlinker.EtherCAT_Master_ATxxxx.Beckhoff_ATH2xxx.Beckhoff_ATH2xxxEK1122.A_0003_ATH2000_0250_0024.CC_Outputs.Current_setpoint_value_Ch[1] <-> CC Outputs/Current setpoint value Ch.2
//     PlcTask Outputs/GVL_iXlinker.EtherCAT_Master_ATxxxx.Beckhoff_ATH2xxx.Beckhoff_ATH2xxxEK1122.A_0003_ATH2000_0250_0024.CC_Outputs.Current_setpoint_value_Ch[2] <-> CC Outputs/Current setpoint value Ch.3
//     PlcTask Outputs/GVL_iXlinker.EtherCAT_Master_ATxxxx.Beckhoff_ATH2xxx.Beckhoff_ATH2xxxEK1122.A_0003_ATH2000_0250_0024.CC_Outputs.Current_setpoint_value_Ch[3] <-> CC Outputs/Current setpoint value Ch.4
//     PlcTask Outputs/GVL_iXlinker.EtherCAT_Master_ATxxxx.Beckhoff_ATH2xxx.Beckhoff_ATH2xxxEK1122.A_0003_ATH2000_0250_0024.CC_Outputs.Current_setpoint_value_Ch[4] <-> CC Outputs/Current setpoint value Ch.5
//     PlcTask Outputs/GVL_iXlinker.EtherCAT_Master_ATxxxx.Beckhoff_ATH2xxx.Beckhoff_ATH2xxxEK1122.A_0003_ATH2000_0250_0024.CC_Outputs.Current_setpoint_value_Ch[5] <-> CC Outputs/Current setpoint value Ch.6
//     PlcTask Outputs/GVL_iXlinker.EtherCAT_Master_ATxxxx.Beckhoff_ATH2xxx.Beckhoff_ATH2xxxEK1122.A_0003_ATH2000_0250_0024.CC_Outputs.Current_setpoint_value_Ch[6] <-> CC Outputs/Current setpoint value Ch.7
//     PlcTask Outputs/GVL_iXlinker.EtherCAT_Master_ATxxxx.Beckhoff_ATH2xxx.Beckhoff_ATH2xxxEK1122.A_0003_ATH2000_0250_0024.CC_Outputs.Current_setpoint_value_Ch[7] <-> CC Outputs/Current setpoint value Ch.8
//     PlcTask Outputs/GVL_iXlinker.EtherCAT_Master_ATxxxx.Beckhoff_ATH2xxx.Beckhoff_ATH2xxxEK1122.A_0003_ATH2000_0250_0024.CC_Outputs.Current_setpoint_value_Ch[8] <-> CC Outputs/Current setpoint value Ch.9
//     PlcTask Outputs/GVL_iXlinker.EtherCAT_Master_ATxxxx.Beckhoff_ATH2xxx.Beckhoff_ATH2xxxEK1122.A_0003_ATH2000_0250_0024.CC_Outputs.Current_setpoint_value_Ch[9] <-> CC Outputs/Current setpoint value Ch.10
//     PlcTask Outputs/GVL_iXlinker.EtherCAT_Master_ATxxxx.Beckhoff_ATH2xxx.Beckhoff_ATH2xxxEK1122.A_0003_ATH2000_0250_0024.CC_Outputs.Current_setpoint_value_Ch[10] <-> CC Outputs/Current setpoint value Ch.11
//     PlcTask Outputs/GVL_iXlinker.EtherCAT_Master_ATxxxx.Beckhoff_ATH2xxx.Beckhoff_ATH2xxxEK1122.A_0003_ATH2000_0250_0024.CC_Outputs.Current_setpoint_value_Ch[11] <-> CC Outputs/Current setpoint value Ch.12
//     PlcTask Outputs/GVL_iXlinker.EtherCAT_Master_ATxxxx.Beckhoff_ATH2xxx.Beckhoff_ATH2xxxEK1122.A_0003_ATH2000_0250_0024.CC_Outputs.Current_setpoint_value_Ch[12] <-> CC Outputs/Current setpoint value Ch.13
//     PlcTask Outputs/GVL_iXlinker.EtherCAT_Master_ATxxxx.Beckhoff_ATH2xxx.Beckhoff_ATH2xxxEK1122.A_0003_ATH2000_0250_0024.CC_Outputs.Current_setpoint_value_Ch[13] <-> CC Outputs/Current setpoint value Ch.14
//     PlcTask Outputs/GVL_iXlinker.EtherCAT_Master_ATxxxx.Beckhoff_ATH2xxx.Beckhoff_ATH2xxxEK1122.A_0003_ATH2000_0250_0024.CC_Outputs.Current_setpoint_value_Ch[14] <-> CC Outputs/Current setpoint value Ch.15
//     PlcTask Inputs/GVL_iXlinker.EtherCAT_Master_ATxxxx.Beckhoff_ATH2xxx.Beckhoff_ATH2xxxEK1122.A_0003_ATH2000_0250_0024.WcState.WcState <-> WcState/WcState
//     PlcTask Inputs/GVL_iXlinker.EtherCAT_Master_ATxxxx.Beckhoff_ATH2xxx.Beckhoff_ATH2xxxEK1122.A_0003_ATH2000_0250_0024.WcState.InputToggle <-> WcState/InputToggle
//     PlcTask Inputs/GVL_iXlinker.EtherCAT_Master_ATxxxx.Beckhoff_ATH2xxx.Beckhoff_ATH2xxxEK1122.A_0003_ATH2000_0250_0024.InfoData.AdsAddr <-> InfoData/AdsAddr
//     PlcTask Inputs/GVL_iXlinker.EtherCAT_Master_ATxxxx.Beckhoff_ATH2xxx.Beckhoff_ATH2xxxEK1122.A_0003_ATH2000_0250_0024.InfoData.DcOutputShift <-> InfoData/DcOutputShift
//     PlcTask Inputs/GVL_iXlinker.EtherCAT_Master_ATxxxx.Beckhoff_ATH2xxx.Beckhoff_ATH2xxxEK1122.A_0003_ATH2000_0250_0024.InfoData.DcInputShift <-> InfoData/DcInputShift
//     PlcTask Inputs/GVL_iXlinker.EtherCAT_Master_ATxxxx.Beckhoff_ATH2xxx.Beckhoff_ATH2xxxEK1122.A_0003_ATH2000_0250_0024.InfoData.State <-> InfoData/State
//   PLC/PLC Instance <-> EtherCAT Master ATxxxx/Beckhoff ATH2xxx/Beckhoff ATH2xxxEK1122/A_0004(ATH2040-0250-0022)
//     PlcTask Inputs/GVL_iXlinker.EtherCAT_Master_ATxxxx.Beckhoff_ATH2xxx.Beckhoff_ATH2xxxEK1122.A_0004_ATH2040_0250_0022.CC_Inputs.Status <-> CC Inputs/Status
//     PlcTask Inputs/GVL_iXlinker.EtherCAT_Master_ATxxxx.Beckhoff_ATH2xxx.Beckhoff_ATH2xxxEK1122.A_0004_ATH2040_0250_0022.CC_Inputs.Current_actual_value_Ch[0] <-> CC Inputs/Current actual value Ch.1
//     PlcTask Inputs/GVL_iXlinker.EtherCAT_Master_ATxxxx.Beckhoff_ATH2xxx.Beckhoff_ATH2xxxEK1122.A_0004_ATH2040_0250_0022.CC_Inputs.Current_actual_value_Ch[1] <-> CC Inputs/Current actual value Ch.2
//     PlcTask Inputs/GVL_iXlinker.EtherCAT_Master_ATxxxx.Beckhoff_ATH2xxx.Beckhoff_ATH2xxxEK1122.A_0004_ATH2040_0250_0022.CC_Inputs.Current_actual_value_Ch[2] <-> CC Inputs/Current actual value Ch.3
//     PlcTask Inputs/GVL_iXlinker.EtherCAT_Master_ATxxxx.Beckhoff_ATH2xxx.Beckhoff_ATH2xxxEK1122.A_0004_ATH2040_0250_0022.CC_Inputs.Current_actual_value_Ch[3] <-> CC Inputs/Current actual value Ch.4
//     PlcTask Inputs/GVL_iXlinker.EtherCAT_Master_ATxxxx.Beckhoff_ATH2xxx.Beckhoff_ATH2xxxEK1122.A_0004_ATH2040_0250_0022.CC_Inputs.Current_actual_value_Ch[4] <-> CC Inputs/Current actual value Ch.5
//     PlcTask Inputs/GVL_iXlinker.EtherCAT_Master_ATxxxx.Beckhoff_ATH2xxx.Beckhoff_ATH2xxxEK1122.A_0004_ATH2040_0250_0022.CC_Inputs.Current_actual_value_Ch[5] <-> CC Inputs/Current actual value Ch.6
//     PlcTask Inputs/GVL_iXlinker.EtherCAT_Master_ATxxxx.Beckhoff_ATH2xxx.Beckhoff_ATH2xxxEK1122.A_0004_ATH2040_0250_0022.CC_Inputs.Current_actual_value_Ch[6] <-> CC Inputs/Current actual value Ch.7
//     PlcTask Inputs/GVL_iXlinker.EtherCAT_Master_ATxxxx.Beckhoff_ATH2xxx.Beckhoff_ATH2xxxEK1122.A_0004_ATH2040_0250_0022.CC_Inputs.Current_actual_value_Ch[7] <-> CC Inputs/Current actual value Ch.8
//     PlcTask Inputs/GVL_iXlinker.EtherCAT_Master_ATxxxx.Beckhoff_ATH2xxx.Beckhoff_ATH2xxxEK1122.A_0004_ATH2040_0250_0022.CC_Inputs.Current_actual_value_Ch[8] <-> CC Inputs/Current actual value Ch.9
//     PlcTask Inputs/GVL_iXlinker.EtherCAT_Master_ATxxxx.Beckhoff_ATH2xxx.Beckhoff_ATH2xxxEK1122.A_0004_ATH2040_0250_0022.CC_Inputs.Current_actual_value_Ch[9] <-> CC Inputs/Current actual value Ch.10
//     PlcTask Inputs/GVL_iXlinker.EtherCAT_Master_ATxxxx.Beckhoff_ATH2xxx.Beckhoff_ATH2xxxEK1122.A_0004_ATH2040_0250_0022.CC_Inputs.Current_actual_value_Ch[10] <-> CC Inputs/Current actual value Ch.11
//     PlcTask Inputs/GVL_iXlinker.EtherCAT_Master_ATxxxx.Beckhoff_ATH2xxx.Beckhoff_ATH2xxxEK1122.A_0004_ATH2040_0250_0022.CC_Inputs.Current_actual_value_Ch[11] <-> CC Inputs/Current actual value Ch.12
//     PlcTask Inputs/GVL_iXlinker.EtherCAT_Master_ATxxxx.Beckhoff_ATH2xxx.Beckhoff_ATH2xxxEK1122.A_0004_ATH2040_0250_0022.CC_Inputs.Current_actual_value_Ch[12] <-> CC Inputs/Current actual value Ch.13
//     PlcTask Inputs/GVL_iXlinker.EtherCAT_Master_ATxxxx.Beckhoff_ATH2xxx.Beckhoff_ATH2xxxEK1122.A_0004_ATH2040_0250_0022.CC_Inputs.Current_actual_value_Ch[13] <-> CC Inputs/Current actual value Ch.14
//     PlcTask Inputs/GVL_iXlinker.EtherCAT_Master_ATxxxx.Beckhoff_ATH2xxx.Beckhoff_ATH2xxxEK1122.A_0004_ATH2040_0250_0022.CC_Inputs.Current_actual_value_Ch[14] <-> CC Inputs/Current actual value Ch.15
//     PlcTask Outputs/GVL_iXlinker.EtherCAT_Master_ATxxxx.Beckhoff_ATH2xxx.Beckhoff_ATH2xxxEK1122.A_0004_ATH2040_0250_0022.CC_Outputs.Control <-> CC Outputs/Control
//     PlcTask Outputs/GVL_iXlinker.EtherCAT_Master_ATxxxx.Beckhoff_ATH2xxx.Beckhoff_ATH2xxxEK1122.A_0004_ATH2040_0250_0022.CC_Outputs.Current_setpoint_value_Ch[0] <-> CC Outputs/Current setpoint value Ch.1
//     PlcTask Outputs/GVL_iXlinker.EtherCAT_Master_ATxxxx.Beckhoff_ATH2xxx.Beckhoff_ATH2xxxEK1122.A_0004_ATH2040_0250_0022.CC_Outputs.Current_setpoint_value_Ch[1] <-> CC Outputs/Current setpoint value Ch.2
//     PlcTask Outputs/GVL_iXlinker.EtherCAT_Master_ATxxxx.Beckhoff_ATH2xxx.Beckhoff_ATH2xxxEK1122.A_0004_ATH2040_0250_0022.CC_Outputs.Current_setpoint_value_Ch[2] <-> CC Outputs/Current setpoint value Ch.3
//     PlcTask Outputs/GVL_iXlinker.EtherCAT_Master_ATxxxx.Beckhoff_ATH2xxx.Beckhoff_ATH2xxxEK1122.A_0004_ATH2040_0250_0022.CC_Outputs.Current_setpoint_value_Ch[3] <-> CC Outputs/Current setpoint value Ch.4
//     PlcTask Outputs/GVL_iXlinker.EtherCAT_Master_ATxxxx.Beckhoff_ATH2xxx.Beckhoff_ATH2xxxEK1122.A_0004_ATH2040_0250_0022.CC_Outputs.Current_setpoint_value_Ch[4] <-> CC Outputs/Current setpoint value Ch.5
//     PlcTask Outputs/GVL_iXlinker.EtherCAT_Master_ATxxxx.Beckhoff_ATH2xxx.Beckhoff_ATH2xxxEK1122.A_0004_ATH2040_0250_0022.CC_Outputs.Current_setpoint_value_Ch[5] <-> CC Outputs/Current setpoint value Ch.6
//     PlcTask Outputs/GVL_iXlinker.EtherCAT_Master_ATxxxx.Beckhoff_ATH2xxx.Beckhoff_ATH2xxxEK1122.A_0004_ATH2040_0250_0022.CC_Outputs.Current_setpoint_value_Ch[6] <-> CC Outputs/Current setpoint value Ch.7
//     PlcTask Outputs/GVL_iXlinker.EtherCAT_Master_ATxxxx.Beckhoff_ATH2xxx.Beckhoff_ATH2xxxEK1122.A_0004_ATH2040_0250_0022.CC_Outputs.Current_setpoint_value_Ch[7] <-> CC Outputs/Current setpoint value Ch.8
//     PlcTask Outputs/GVL_iXlinker.EtherCAT_Master_ATxxxx.Beckhoff_ATH2xxx.Beckhoff_ATH2xxxEK1122.A_0004_ATH2040_0250_0022.CC_Outputs.Current_setpoint_value_Ch[8] <-> CC Outputs/Current setpoint value Ch.9
//     PlcTask Outputs/GVL_iXlinker.EtherCAT_Master_ATxxxx.Beckhoff_ATH2xxx.Beckhoff_ATH2xxxEK1122.A_0004_ATH2040_0250_0022.CC_Outputs.Current_setpoint_value_Ch[9] <-> CC Outputs/Current setpoint value Ch.10
//     PlcTask Outputs/GVL_iXlinker.EtherCAT_Master_ATxxxx.Beckhoff_ATH2xxx.Beckhoff_ATH2xxxEK1122.A_0004_ATH2040_0250_0022.CC_Outputs.Current_setpoint_value_Ch[10] <-> CC Outputs/Current setpoint value Ch.11
//     PlcTask Outputs/GVL_iXlinker.EtherCAT_Master_ATxxxx.Beckhoff_ATH2xxx.Beckhoff_ATH2xxxEK1122.A_0004_ATH2040_0250_0022.CC_Outputs.Current_setpoint_value_Ch[11] <-> CC Outputs/Current setpoint value Ch.12
//     PlcTask Outputs/GVL_iXlinker.EtherCAT_Master_ATxxxx.Beckhoff_ATH2xxx.Beckhoff_ATH2xxxEK1122.A_0004_ATH2040_0250_0022.CC_Outputs.Current_setpoint_value_Ch[12] <-> CC Outputs/Current setpoint value Ch.13
//     PlcTask Outputs/GVL_iXlinker.EtherCAT_Master_ATxxxx.Beckhoff_ATH2xxx.Beckhoff_ATH2xxxEK1122.A_0004_ATH2040_0250_0022.CC_Outputs.Current_setpoint_value_Ch[13] <-> CC Outputs/Current setpoint value Ch.14
//     PlcTask Outputs/GVL_iXlinker.EtherCAT_Master_ATxxxx.Beckhoff_ATH2xxx.Beckhoff_ATH2xxxEK1122.A_0004_ATH2040_0250_0022.CC_Outputs.Current_setpoint_value_Ch[14] <-> CC Outputs/Current setpoint value Ch.15
//     PlcTask Inputs/GVL_iXlinker.EtherCAT_Master_ATxxxx.Beckhoff_ATH2xxx.Beckhoff_ATH2xxxEK1122.A_0004_ATH2040_0250_0022.WcState.WcState <-> WcState/WcState
//     PlcTask Inputs/GVL_iXlinker.EtherCAT_Master_ATxxxx.Beckhoff_ATH2xxx.Beckhoff_ATH2xxxEK1122.A_0004_ATH2040_0250_0022.WcState.InputToggle <-> WcState/InputToggle
//     PlcTask Inputs/GVL_iXlinker.EtherCAT_Master_ATxxxx.Beckhoff_ATH2xxx.Beckhoff_ATH2xxxEK1122.A_0004_ATH2040_0250_0022.InfoData.AdsAddr <-> InfoData/AdsAddr
//     PlcTask Inputs/GVL_iXlinker.EtherCAT_Master_ATxxxx.Beckhoff_ATH2xxx.Beckhoff_ATH2xxxEK1122.A_0004_ATH2040_0250_0022.InfoData.DcOutputShift <-> InfoData/DcOutputShift
//     PlcTask Inputs/GVL_iXlinker.EtherCAT_Master_ATxxxx.Beckhoff_ATH2xxx.Beckhoff_ATH2xxxEK1122.A_0004_ATH2040_0250_0022.InfoData.DcInputShift <-> InfoData/DcInputShift
